LIN {X 0,Y 227.878,Z 329.572,A -85,B 0,C 180,E1 -19946.376,E2 -19946.376} C_VEL
LIN {X 0,Y 227.902,Z 329.591,A -85,B 0,C 180,E1 -19950.434,E2 -19950.434} C_VEL
LIN {X 0,Y 227.922,Z 329.564,A -85,B 0,C 180,E1 -19954.424,E2 -19954.424} C_VEL
LIN {X 0,Y 227.944,Z 329.583,A -85,B 0,C 180,E1 -19958.284,E2 -19958.284} C_VEL
LIN {X 0,Y 228.03,Z 329.545,A -85,B 0,C 180,E1 -19962.826,E2 -19962.826} C_VEL
LIN {X 0,Y 228.067,Z 329.562,A -85,B 0,C 180,E1 -19967.542,E2 -19967.542} C_VEL
LIN {X 0,Y 228.263,Z 329.504,A -85,B 0,C 180,E1 -19971.143,E2 -19971.143} C_VEL
LIN {X 0,Y 228.319,Z 329.521,A -85,B 0,C 180,E1 -19972.926,E2 -19972.926} C_VEL
LIN {X 0,Y 228.549,Z 329.485,A -85,B 0,C 180,E1 -19978.237,E2 -19978.237} C_VEL
LIN {X 0,Y 228.548,Z 329.475,A -85,B 0,C 180,E1 -19981.761,E2 -19981.761} C_VEL
LIN {X 0,Y 228.318,Z 329.531,A -85,B 0,C 180,E1 -19987.072,E2 -19987.072} C_VEL
LIN {X 0,Y 228.14,Z 329.521,A -85,B 0,C 180,E1 -19990.65,E2 -19990.65} C_VEL
LIN {X 0,Y 228.057,Z 329.576,A -85,B 0,C 180,E1 -19994.272,E2 -19994.272} C_VEL
LIN {X 0,Y 227.997,Z 329.55,A -85,B 0,C 180,E1 -19997.953,E2 -19997.953} C_VEL
LIN {X 0,Y 227.924,Z 329.589,A -85,B 0,C 180,E1 -20002.329,E2 -20002.329} C_VEL
LIN {X 0,Y 227.936,Z 329.561,A -85,B 0,C 180,E1 -20006.602,E2 -20006.602} C_VEL
LIN {X 0,Y 227.891,Z 329.596,A -85,B 0,C 180,E1 -20010.291,E2 -20010.291} C_VEL
LIN {X 0,Y 227.884,Z 329.576,A -85,B 0,C 180,E1 -20013.718,E2 -20013.718} C_VEL
LIN {X 0,Y 227.866,Z 329.604,A -85,B 0,C 180,E1 -20018.085,E2 -20018.085} C_VEL
LIN {X 0,Y 227.904,Z 329.593,A -85,B 0,C 180,E1 -20022.719,E2 -20022.719} C_VEL
LIN {X 0,Y 227.815,Z 329.543,A -85,B 0,C 180,E1 -20027.26,E2 -20027.26} C_VEL
LIN {X 0,Y 227.865,Z 329.603,A -85,B 0,C 180,E1 -20031.914,E2 -20031.914} C_VEL
LIN {X 0,Y 227.948,Z 329.901,A -85,B 0,C 180,E1 -20032.928,E2 -20032.928} C_VEL
LIN {X 0,Y 228.323,Z 331.21,A -85,B 0,C 180,E1 -20033.243,E2 -20033.243} C_VEL
LIN {X 0,Y 229.942,Z 333.723,A -85,B 0,C 180,E1 -20033.654,E2 -20033.654} C_VEL
LIN {X 0,Y 238.78,Z 348.968,A -85,B 0,C 180,E1 -20035.756,E2 -20035.756} C_VEL
LIN {X 0,Y 244.929,Z 360.706,A -85,B 0,C 180,E1 -20037.14,E2 -20037.14} C_VEL
LIN {X 0,Y 252.144,Z 374.306,A -85,B 0,C 180,E1 -20038.647,E2 -20038.647} C_VEL
LIN {X 0,Y 260.818,Z 387.178,A -85,B 0,C 180,E1 -20040.211,E2 -20040.211} C_VEL
LIN {X 0,Y 271.78,Z 400.26,A -85,B 0,C 180,E1 -20041.921,E2 -20041.921} C_VEL
LIN {X 0,Y 286.362,Z 414.958,A -85,B 0,C 180,E1 -20043.882,E2 -20043.882} C_VEL
LIN {X 0,Y 299.444,Z 426.122,A -85,B 0,C 180,E1 -20045.43,E2 -20045.43} C_VEL
LIN {X 0,Y 307.549,Z 432.734,A -85,B 0,C 180,E1 -20046.478,E2 -20046.478} C_VEL
LIN {X 0,Y 315.593,Z 438.951,A -85,B 0,C 180,E1 -20047.734,E2 -20047.734} C_VEL
LIN {X 0,Y 323.402,Z 444.777,A -85,B 0,C 180,E1 -20049.138,E2 -20049.138} C_VEL
LIN {X 0,Y 331.993,Z 451.224,A -85,B 0,C 180,E1 -20050.908,E2 -20050.908} C_VEL
LIN {X 0,Y 339.546,Z 456.264,A -85,B 0,C 180,E1 -20052.64,E2 -20052.64} C_VEL
LIN {X 0,Y 346.066,Z 461.128,A -85,B 0,C 180,E1 -20054.389,E2 -20054.389} C_VEL
LIN {X 0,Y 351.939,Z 464.834,A -85,B 0,C 180,E1 -20056.135,E2 -20056.135} C_VEL
LIN {X 0,Y 355.953,Z 467.098,A -85,B 0,C 180,E1 -20057.457,E2 -20057.457} C_VEL
LIN {X 0,Y 359.121,Z 469.614,A -85,B 0,C 180,E1 -20058.715,E2 -20058.715} C_VEL
LIN {X 0,Y 363.316,Z 472.458,A -85,B 0,C 180,E1 -20060.586,E2 -20060.586} C_VEL
LIN {X 0,Y 366.572,Z 474.299,A -85,B 0,C 180,E1 -20062.288,E2 -20062.288} C_VEL
LIN {X 0,Y 368.408,Z 475.23,A -85,B 0,C 180,E1 -20063.428,E2 -20063.428} C_VEL
LIN {X 0,Y 369.974,Z 475.879,A -85,B 0,C 180,E1 -20064.55,E2 -20064.55} C_VEL
LIN {X 0,Y 371.244,Z 476.349,A -85,B 0,C 180,E1 -20065.657,E2 -20065.657} C_VEL
LIN {X 0,Y 372.236,Z 476.635,A -85,B 0,C 180,E1 -20066.753,E2 -20066.753} C_VEL
LIN {X 0,Y 372.866,Z 477.016,A -85,B 0,C 180,E1 -20067.84,E2 -20067.84} C_VEL
LIN {X 0,Y 373.24,Z 477.247,A -85,B 0,C 180,E1 -20068.921,E2 -20068.921} C_VEL
LIN {X 0,Y 373.406,Z 477.203,A -85,B 0,C 180,E1 -20070,E2 -20070} C_VEL
LIN {X 0,Y 373.262,Z 477.182,A -85,B 0,C 180,E1 -20071.079,E2 -20071.079} C_VEL
LIN {X 0,Y 372.799,Z 476.9,A -85,B 0,C 180,E1 -20072.374,E2 -20072.374} C_VEL
LIN {X 0,Y 371.247,Z 476.345,A -85,B 0,C 180,E1 -20074.343,E2 -20074.343} C_VEL
LIN {X 0,Y 369.982,Z 475.883,A -85,B 0,C 180,E1 -20075.45,E2 -20075.45} C_VEL
LIN {X 0,Y 368.059,Z 475.041,A -85,B 0,C 180,E1 -20076.825,E2 -20076.825} C_VEL
LIN {X 0,Y 366.576,Z 474.352,A -85,B 0,C 180,E1 -20077.712,E2 -20077.712} C_VEL
LIN {X 0,Y 363.307,Z 472.462,A -85,B 0,C 180,E1 -20079.406,E2 -20079.406} C_VEL
LIN {X 0,Y 359.105,Z 469.613,A -85,B 0,C 180,E1 -20081.286,E2 -20081.286} C_VEL
LIN {X 0,Y 355.912,Z 467.07,A -85,B 0,C 180,E1 -20082.545,E2 -20082.545} C_VEL
LIN {X 0,Y 351.918,Z 464.861,A -85,B 0,C 180,E1 -20083.865,E2 -20083.865} C_VEL
LIN {X 0,Y 345.56,Z 460.756,A -85,B 0,C 180,E1 -20085.755,E2 -20085.755} C_VEL
LIN {X 0,Y 338.472,Z 455.62,A -85,B 0,C 180,E1 -20087.612,E2 -20087.612} C_VEL
LIN {X 0,Y 330.629,Z 450.246,A -85,B 0,C 180,E1 -20089.388,E2 -20089.388} C_VEL
LIN {X 0,Y 323.191,Z 444.661,A -85,B 0,C 180,E1 -20090.898,E2 -20090.898} C_VEL
LIN {X 0,Y 315.18,Z 438.628,A -85,B 0,C 180,E1 -20092.332,E2 -20092.332} C_VEL
LIN {X 0,Y 306.65,Z 432.052,A -85,B 0,C 180,E1 -20093.65,E2 -20093.65} C_VEL
LIN {X 0,Y 297.197,Z 424.33,A -85,B 0,C 180,E1 -20094.843,E2 -20094.843} C_VEL
LIN {X 0,Y 282.743,Z 411.497,A -85,B 0,C 180,E1 -20096.577,E2 -20096.577} C_VEL
LIN {X 0,Y 269.021,Z 397.22,A -85,B 0,C 180,E1 -20098.486,E2 -20098.486} C_VEL
LIN {X 0,Y 260.299,Z 386.445,A -85,B 0,C 180,E1 -20099.878,E2 -20099.878} C_VEL
LIN {X 0,Y 252.01,Z 374.071,A -85,B 0,C 180,E1 -20101.38,E2 -20101.38} C_VEL
LIN {X 0,Y 245.107,Z 361.073,A -85,B 0,C 180,E1 -20102.82,E2 -20102.82} C_VEL
LIN {X 0,Y 239.021,Z 349.422,A -85,B 0,C 180,E1 -20104.188,E2 -20104.188} C_VEL
LIN {X 0,Y 231.592,Z 336.596,A -85,B 0,C 180,E1 -20105.936,E2 -20105.936} C_VEL
LIN {X 0,Y 229.583,Z 333.337,A -85,B 0,C 180,E1 -20106.427,E2 -20106.427} C_VEL
LIN {X 0,Y 228.039,Z 330.419,A -85,B 0,C 180,E1 -20106.894,E2 -20106.894} C_VEL
LIN {X 0,Y 227.9,Z 329.657,A -85,B 0,C 180,E1 -20107.311,E2 -20107.311} C_VEL
LIN {X 0,Y 227.83,Z 329.551,A -85,B 0,C 180,E1 -20110.375,E2 -20110.375} C_VEL
LIN {X 0,Y 227.852,Z 329.579,A -85,B 0,C 180,E1 -20115.187,E2 -20115.187} C_VEL
LIN {X 0,Y 227.904,Z 329.586,A -85,B 0,C 180,E1 -20117.739,E2 -20117.739} C_VEL
LIN {X 0,Y 227.866,Z 329.604,A -85,B 0,C 180,E1 -20121.915,E2 -20121.915} C_VEL
LIN {X 0,Y 227.884,Z 329.576,A -85,B 0,C 180,E1 -20126.374,E2 -20126.374} C_VEL
LIN {X 0,Y 227.898,Z 329.583,A -85,B 0,C 180,E1 -20130.436,E2 -20130.436} C_VEL
LIN {X 0,Y 227.923,Z 329.574,A -85,B 0,C 180,E1 -20134.426,E2 -20134.426} C_VEL
LIN {X 0,Y 227.956,Z 329.575,A -85,B 0,C 180,E1 -20138.288,E2 -20138.288} C_VEL
LIN {X 0,Y 228.029,Z 329.557,A -85,B 0,C 180,E1 -20142.827,E2 -20142.827} C_VEL
LIN {X 0,Y 228.066,Z 329.554,A -85,B 0,C 180,E1 -20147.544,E2 -20147.544} C_VEL
LIN {X 0,Y 228.261,Z 329.51,A -85,B 0,C 180,E1 -20151.145,E2 -20151.145} C_VEL
LIN {X 0,Y 228.318,Z 329.531,A -85,B 0,C 180,E1 -20152.928,E2 -20152.928} C_VEL
LIN {X 0,Y 228.548,Z 329.475,A -85,B 0,C 180,E1 -20158.239,E2 -20158.239} C_VEL
LIN {X 0,Y 228.549,Z 329.485,A -85,B 0,C 180,E1 -20161.763,E2 -20161.763} C_VEL
LIN {X 0,Y 228.319,Z 329.521,A -85,B 0,C 180,E1 -20167.074,E2 -20167.074} C_VEL
LIN {X 0,Y 228.141,Z 329.523,A -85,B 0,C 180,E1 -20170.652,E2 -20170.652} C_VEL
LIN {X 0,Y 228.056,Z 329.575,A -85,B 0,C 180,E1 -20174.274,E2 -20174.274} C_VEL
LIN {X 0,Y 227.998,Z 329.542,A -85,B 0,C 180,E1 -20177.955,E2 -20177.955} C_VEL
LIN {X 0,Y 227.914,Z 329.591,A -85,B 0,C 180,E1 -20182.322,E2 -20182.322} C_VEL
LIN {X 0,Y 227.939,Z 329.556,A -85,B 0,C 180,E1 -20186.603,E2 -20186.603} C_VEL
LIN {X 0,Y 227.895,Z 329.597,A -85,B 0,C 180,E1 -20190.292,E2 -20190.292} C_VEL
LIN {X 0,Y 227.876,Z 329.572,A -85,B 0,C 180,E1 -20193.722,E2 -20193.722} C_VEL
LIN {X 0,Y 227.842,Z 329.599,A -85,B 0,C 180,E1 -20198.093,E2 -20198.093} C_VEL
LIN {X 0,Y 227.803,Z 329.608,A -85,B 0,C 180,E1 -20202.746,E2 -20202.746} C_VEL
LIN {X 0,Y 227.825,Z 329.62,A -85,B 0,C 180,E1 -20207.425,E2 -20207.425} C_VEL
LIN {X 0,Y 229.604,Z 337.052,A -85,B 0,C 180,E1 -20212.253,E2 -20212.253} C_VEL
LIN {X 0,Y 230.128,Z 339.355,A -85,B 0,C 180,E1 -20213.453,E2 -20213.453} C_VEL
LIN {X 0,Y 232.001,Z 343.344,A -85,B 0,C 180,E1 -20214.006,E2 -20214.006} C_VEL
LIN {X 0,Y 238.477,Z 356.937,A -85,B 0,C 180,E1 -20215.607,E2 -20215.607} C_VEL
LIN {X 0,Y 243.683,Z 369.149,A -85,B 0,C 180,E1 -20216.856,E2 -20216.856} C_VEL
LIN {X 0,Y 247.391,Z 390.036,A -85,B 0,C 180,E1 -20218.112,E2 -20218.112} C_VEL
LIN {X 0,Y 248.128,Z 394.813,A -85,B 0,C 180,E1 -20218.376,E2 -20218.376} C_VEL
LIN {X 0,Y 248.036,Z 398.357,A -85,B 0,C 180,E1 -20218.48,E2 -20218.48} C_VEL
LIN {X 0,Y 247.212,Z 404.208,A -85,B 0,C 180,E1 -20218.559,E2 -20218.559} C_VEL
LIN {X 0,Y 241.542,Z 423.223,A -85,B 0,C 180,E1 -20218.39,E2 -20218.39} C_VEL
LIN {X 0,Y 240.791,Z 429.07,A -85,B 0,C 180,E1 -20218.481,E2 -20218.481} C_VEL
LIN {X 0,Y 239.894,Z 448.706,A -85,B 0,C 180,E1 -20219.122,E2 -20219.122} C_VEL
LIN {X 0,Y 238.364,Z 462.733,A -85,B 0,C 180,E1 -20219.919,E2 -20219.919} C_VEL
LIN {X 0,Y 236.772,Z 473.371,A -85,B 0,C 180,E1 -20220.798,E2 -20220.798} C_VEL
LIN {X 0,Y 234.904,Z 483.507,A -85,B 0,C 180,E1 -20221.887,E2 -20221.887} C_VEL
LIN {X 0,Y 232.976,Z 492.498,A -85,B 0,C 180,E1 -20223.097,E2 -20223.097} C_VEL
LIN {X 0,Y 230.911,Z 501.222,A -85,B 0,C 180,E1 -20224.539,E2 -20224.539} C_VEL
LIN {X 0,Y 228.989,Z 508.613,A -85,B 0,C 180,E1 -20226.005,E2 -20226.005} C_VEL
LIN {X 0,Y 227.036,Z 515.83,A -85,B 0,C 180,E1 -20227.716,E2 -20227.716} C_VEL
LIN {X 0,Y 225.39,Z 522.16,A -85,B 0,C 180,E1 -20229.508,E2 -20229.508} C_VEL
LIN {X 0,Y 223.506,Z 528.569,A -85,B 0,C 180,E1 -20231.673,E2 -20231.673} C_VEL
LIN {X 0,Y 222.258,Z 533.072,A -85,B 0,C 180,E1 -20233.466,E2 -20233.466} C_VEL
LIN {X 0,Y 220.614,Z 538.563,A -85,B 0,C 180,E1 -20236.177,E2 -20236.177} C_VEL
LIN {X 0,Y 219.59,Z 542.893,A -85,B 0,C 180,E1 -20238.929,E2 -20238.929} C_VEL
LIN {X 0,Y 219.09,Z 545.263,A -85,B 0,C 180,E1 -20240.771,E2 -20240.771} C_VEL
LIN {X 0,Y 218.738,Z 547.065,A -85,B 0,C 180,E1 -20242.616,E2 -20242.616} C_VEL
LIN {X 0,Y 218.501,Z 549.519,A -85,B 0,C 180,E1 -20246.312,E2 -20246.312} C_VEL
LIN {X 0,Y 218.525,Z 550.112,A -85,B 0,C 180,E1 -20248.157,E2 -20248.157} C_VEL
LIN {X 0,Y 218.623,Z 550.27,A -85,B 0,C 180,E1 -20250,E2 -20250} C_VEL
LIN {X 0,Y 218.524,Z 550.112,A -85,B 0,C 180,E1 -20251.843,E2 -20251.843} C_VEL
LIN {X 0,Y 218.484,Z 549.256,A -85,B 0,C 180,E1 -20254.292,E2 -20254.292} C_VEL
LIN {X 0,Y 218.711,Z 547.064,A -85,B 0,C 180,E1 -20257.385,E2 -20257.385} C_VEL
LIN {X 0,Y 219.319,Z 544.111,A -85,B 0,C 180,E1 -20260.151,E2 -20260.151} C_VEL
LIN {X 0,Y 220.226,Z 540.118,A -85,B 0,C 180,E1 -20262.908,E2 -20262.908} C_VEL
LIN {X 0,Y 221.657,Z 534.987,A -85,B 0,C 180,E1 -20265.635,E2 -20265.635} C_VEL
LIN {X 0,Y 223.184,Z 529.726,A -85,B 0,C 180,E1 -20267.88,E2 -20267.88} C_VEL
LIN {X 0,Y 225.063,Z 523.411,A -85,B 0,C 180,E1 -20270.089,E2 -20270.089} C_VEL
LIN {X 0,Y 226.621,Z 517.457,A -85,B 0,C 180,E1 -20271.847,E2 -20271.847} C_VEL
LIN {X 0,Y 228.474,Z 510.531,A -85,B 0,C 180,E1 -20273.571,E2 -20273.571} C_VEL
LIN {X 0,Y 230.658,Z 502.357,A -85,B 0,C 180,E1 -20275.249,E2 -20275.249} C_VEL
LIN {X 0,Y 232.662,Z 493.849,A -85,B 0,C 180,E1 -20276.7,E2 -20276.7} C_VEL
LIN {X 0,Y 234.592,Z 485.139,A -85,B 0,C 180,E1 -20277.91,E2 -20277.91} C_VEL
LIN {X 0,Y 236.374,Z 475.383,A -85,B 0,C 180,E1 -20279.012,E2 -20279.012} C_VEL
LIN {X 0,Y 237.76,Z 466.593,A -85,B 0,C 180,E1 -20279.799,E2 -20279.799} C_VEL
LIN {X 0,Y 239.164,Z 456.049,A -85,B 0,C 180,E1 -20280.5,E2 -20280.5} C_VEL
LIN {X 0,Y 240.048,Z 446.427,A -85,B 0,C 180,E1 -20280.96,E2 -20280.96} C_VEL
LIN {X 0,Y 241.421,Z 414.37,A -85,B 0,C 180,E1 -20281.93,E2 -20281.93} C_VEL
LIN {X 0,Y 242.009,Z 395.189,A -85,B 0,C 180,E1 -20282.501,E2 -20282.501} C_VEL
LIN {X 0,Y 238.137,Z 372.45,A -85,B 0,C 180,E1 -20283.896,E2 -20283.896} C_VEL
LIN {X 0,Y 232.185,Z 358.251,A -85,B 0,C 180,E1 -20285.406,E2 -20285.406} C_VEL
LIN {X 0,Y 224.648,Z 342.853,A -85,B 0,C 180,E1 -20287.378,E2 -20287.378} C_VEL
LIN {X 0,Y 222.799,Z 338.923,A -85,B 0,C 180,E1 -20288.001,E2 -20288.001} C_VEL
LIN {X 0,Y 221.282,Z 332.871,A -85,B 0,C 180,E1 -20291.832,E2 -20291.832} C_VEL
LIN {X 0,Y 220.752,Z 330.49,A -85,B 0,C 180,E1 -20293.611,E2 -20293.611} C_VEL
LIN {X 0,Y 220.762,Z 330.485,A -85,B 0,C 180,E1 -20298.044,E2 -20298.044} C_VEL
LIN {X 0,Y 220.824,Z 330.479,A -85,B 0,C 180,E1 -20302.792,E2 -20302.792} C_VEL
LIN {X 0,Y 220.815,Z 330.458,A -85,B 0,C 180,E1 -20307.242,E2 -20307.242} C_VEL
LIN {X 0,Y 220.824,Z 330.454,A -85,B 0,C 180,E1 -20311.484,E2 -20311.484} C_VEL
LIN {X 0,Y 220.859,Z 330.46,A -85,B 0,C 180,E1 -20315.563,E2 -20315.563} C_VEL
LIN {X 0,Y 220.88,Z 330.442,A -85,B 0,C 180,E1 -20319.512,E2 -20319.512} C_VEL
LIN {X 0,Y 221.011,Z 330.426,A -85,B 0,C 180,E1 -20323.369,E2 -20323.369} C_VEL
LIN {X 0,Y 221.006,Z 330.445,A -85,B 0,C 180,E1 -20327.137,E2 -20327.137} C_VEL
LIN {X 0,Y 221.2,Z 330.382,A -85,B 0,C 180,E1 -20330.858,E2 -20330.858} C_VEL
LIN {X 0,Y 221.254,Z 330.395,A -85,B 0,C 180,E1 -20332.699,E2 -20332.699} C_VEL
LIN {X 0,Y 221.507,Z 330.361,A -85,B 0,C 180,E1 -20338.181,E2 -20338.181} C_VEL
LIN {X 0,Y 221.506,Z 330.352,A -85,B 0,C 180,E1 -20341.817,E2 -20341.817} C_VEL
LIN {X 0,Y 221.253,Z 330.407,A -85,B 0,C 180,E1 -20347.299,E2 -20347.299} C_VEL
LIN {X 0,Y 221.062,Z 330.404,A -85,B 0,C 180,E1 -20350.996,E2 -20350.996} C_VEL
LIN {X 0,Y 220.989,Z 330.459,A -85,B 0,C 180,E1 -20354.738,E2 -20354.738} C_VEL
LIN {X 0,Y 220.916,Z 330.427,A -85,B 0,C 180,E1 -20358.549,E2 -20358.549} C_VEL
LIN {X 0,Y 220.891,Z 330.467,A -85,B 0,C 180,E1 -20362.682,E2 -20362.682} C_VEL
LIN {X 0,Y 220.878,Z 330.437,A -85,B 0,C 180,E1 -20367.014,E2 -20367.014} C_VEL
LIN {X 0,Y 220.833,Z 330.478,A -85,B 0,C 180,E1 -20370.767,E2 -20370.767} C_VEL
LIN {X 0,Y 220.81,Z 330.454,A -85,B 0,C 180,E1 -20374.952,E2 -20374.952} C_VEL
LIN {X 0,Y 220.851,Z 330.459,A -85,B 0,C 180,E1 -20379.526,E2 -20379.526} C_VEL
LIN {X 0,Y 220.861,Z 330.472,A -85,B 0,C 180,E1 -20382.957,E2 -20382.957} C_VEL
LIN {X 0,Y 220.774,Z 330.417,A -85,B 0,C 180,E1 -20388.05,E2 -20388.05} C_VEL
LIN {X 0,Y 220.834,Z 330.704,A -85,B 0,C 180,E1 -20391.492,E2 -20391.492} C_VEL
LIN {X 0,Y 221.134,Z 331.799,A -85,B 0,C 180,E1 -20391.846,E2 -20391.846} C_VEL
LIN {X 0,Y 222.663,Z 334.447,A -85,B 0,C 180,E1 -20392.282,E2 -20392.282} C_VEL
LIN {X 0,Y 223.911,Z 336.348,A -85,B 0,C 180,E1 -20392.606,E2 -20392.606} C_VEL
LIN {X 0,Y 230.101,Z 346.534,A -85,B 0,C 180,E1 -20394.169,E2 -20394.169} C_VEL
LIN {X 0,Y 237.952,Z 360.997,A -85,B 0,C 180,E1 -20396.05,E2 -20396.05} C_VEL
LIN {X 0,Y 246.369,Z 377.37,A -85,B 0,C 180,E1 -20397.922,E2 -20397.922} C_VEL
LIN {X 0,Y 254.153,Z 389.318,A -85,B 0,C 180,E1 -20399.409,E2 -20399.409} C_VEL
LIN {X 0,Y 261.639,Z 398.978,A -85,B 0,C 180,E1 -20400.68,E2 -20400.68} C_VEL
LIN {X 0,Y 273.729,Z 412.316,A -85,B 0,C 180,E1 -20402.491,E2 -20402.491} C_VEL
LIN {X 0,Y 285.746,Z 423.639,A -85,B 0,C 180,E1 -20404.059,E2 -20404.059} C_VEL
LIN {X 0,Y 296.322,Z 432.546,A -85,B 0,C 180,E1 -20405.321,E2 -20405.321} C_VEL
LIN {X 0,Y 304.747,Z 439.439,A -85,B 0,C 180,E1 -20406.447,E2 -20406.447} C_VEL
LIN {X 0,Y 312.979,Z 445.791,A -85,B 0,C 180,E1 -20407.749,E2 -20407.749} C_VEL
LIN {X 0,Y 321.068,Z 451.705,A -85,B 0,C 180,E1 -20409.206,E2 -20409.206} C_VEL
LIN {X 0,Y 329.282,Z 457.928,A -85,B 0,C 180,E1 -20410.918,E2 -20410.918} C_VEL
LIN {X 0,Y 335.929,Z 462.269,A -85,B 0,C 180,E1 -20412.432,E2 -20412.432} C_VEL
LIN {X 0,Y 343.054,Z 467.541,A -85,B 0,C 180,E1 -20414.335,E2 -20414.335} C_VEL
LIN {X 0,Y 348.712,Z 471.122,A -85,B 0,C 180,E1 -20416.005,E2 -20416.005} C_VEL
LIN {X 0,Y 352.903,Z 473.494,A -85,B 0,C 180,E1 -20417.372,E2 -20417.372} C_VEL
LIN {X 0,Y 357.621,Z 477.083,A -85,B 0,C 180,E1 -20419.293,E2 -20419.293} C_VEL
LIN {X 0,Y 361.361,Z 479.527,A -85,B 0,C 180,E1 -20421.049,E2 -20421.049} C_VEL
LIN {X 0,Y 363.554,Z 480.72,A -85,B 0,C 180,E1 -20422.223,E2 -20422.223} C_VEL
LIN {X 0,Y 365.437,Z 481.66,A -85,B 0,C 180,E1 -20423.374,E2 -20423.374} C_VEL
LIN {X 0,Y 367.106,Z 482.343,A -85,B 0,C 180,E1 -20424.558,E2 -20424.558} C_VEL
LIN {X 0,Y 368.313,Z 482.82,A -85,B 0,C 180,E1 -20425.623,E2 -20425.623} C_VEL
LIN {X 0,Y 369.336,Z 483.098,A -85,B 0,C 180,E1 -20426.728,E2 -20426.728} C_VEL
LIN {X 0,Y 369.975,Z 483.474,A -85,B 0,C 180,E1 -20427.823,E2 -20427.823} C_VEL
LIN {X 0,Y 370.339,Z 483.726,A -85,B 0,C 180,E1 -20428.913,E2 -20428.913} C_VEL
LIN {X 0,Y 370.525,Z 483.663,A -85,B 0,C 180,E1 -20430,E2 -20430} C_VEL
LIN {X 0,Y 370.371,Z 483.642,A -85,B 0,C 180,E1 -20431.087,E2 -20431.087} C_VEL
LIN {X 0,Y 369.987,Z 483.423,A -85,B 0,C 180,E1 -20432.177,E2 -20432.177} C_VEL
LIN {X 0,Y 369.321,Z 483.102,A -85,B 0,C 180,E1 -20433.273,E2 -20433.273} C_VEL
LIN {X 0,Y 368.31,Z 482.8,A -85,B 0,C 180,E1 -20434.377,E2 -20434.377} C_VEL
LIN {X 0,Y 367.031,Z 482.313,A -85,B 0,C 180,E1 -20435.494,E2 -20435.494} C_VEL
LIN {X 0,Y 365.444,Z 481.652,A -85,B 0,C 180,E1 -20436.626,E2 -20436.626} C_VEL
LIN {X 0,Y 362.343,Z 480.064,A -85,B 0,C 180,E1 -20438.435,E2 -20438.435} C_VEL
LIN {X 0,Y 358.865,Z 477.939,A -85,B 0,C 180,E1 -20440.151,E2 -20440.151} C_VEL
LIN {X 0,Y 354.945,Z 475.149,A -85,B 0,C 180,E1 -20441.816,E2 -20441.816} C_VEL
LIN {X 0,Y 352.819,Z 473.432,A -85,B 0,C 180,E1 -20442.657,E2 -20442.657} C_VEL
LIN {X 0,Y 347.994,Z 470.716,A -85,B 0,C 180,E1 -20444.215,E2 -20444.215} C_VEL
LIN {X 0,Y 343.051,Z 467.515,A -85,B 0,C 180,E1 -20445.664,E2 -20445.664} C_VEL
LIN {X 0,Y 338.092,Z 463.919,A -85,B 0,C 180,E1 -20447.021,E2 -20447.021} C_VEL
LIN {X 0,Y 330.724,Z 458.91,A -85,B 0,C 180,E1 -20448.764,E2 -20448.764} C_VEL
LIN {X 0,Y 323.285,Z 453.33,A -85,B 0,C 180,E1 -20450.354,E2 -20450.354} C_VEL
LIN {X 0,Y 314.631,Z 447.083,A -85,B 0,C 180,E1 -20451.967,E2 -20451.967} C_VEL
LIN {X 0,Y 306.173,Z 440.522,A -85,B 0,C 180,E1 -20453.342,E2 -20453.342} C_VEL
LIN {X 0,Y 298.373,Z 434.289,A -85,B 0,C 180,E1 -20454.424,E2 -20454.424} C_VEL
LIN {X 0,Y 286.312,Z 424.127,A -85,B 0,C 180,E1 -20455.872,E2 -20455.872} C_VEL
LIN {X 0,Y 276.694,Z 415.179,A -85,B 0,C 180,E1 -20457.106,E2 -20457.106} C_VEL
LIN {X 0,Y 264.358,Z 402.242,A -85,B 0,C 180,E1 -20458.887,E2 -20458.887} C_VEL
LIN {X 0,Y 255.511,Z 391.242,A -85,B 0,C 180,E1 -20460.348,E2 -20460.348} C_VEL
LIN {X 0,Y 247.05,Z 378.539,A -85,B 0,C 180,E1 -20461.939,E2 -20461.939} C_VEL
LIN {X 0,Y 240.025,Z 365.188,A -85,B 0,C 180,E1 -20463.467,E2 -20463.467} C_VEL
LIN {X 0,Y 232.852,Z 351.396,A -85,B 0,C 180,E1 -20465.16,E2 -20465.16} C_VEL
LIN {X 0,Y 225.32,Z 338.515,A -85,B 0,C 180,E1 -20467.034,E2 -20467.034} C_VEL
LIN {X 0,Y 222.666,Z 334.413,A -85,B 0,C 180,E1 -20467.718,E2 -20467.718} C_VEL
LIN {X 0,Y 221.134,Z 331.801,A -85,B 0,C 180,E1 -20468.154,E2 -20468.154} C_VEL
LIN {X 0,Y 220.855,Z 330.69,A -85,B 0,C 180,E1 -20468.515,E2 -20468.515} C_VEL
LIN {X 0,Y 220.774,Z 330.417,A -85,B 0,C 180,E1 -20471.95,E2 -20471.95} C_VEL
LIN {X 0,Y 220.861,Z 330.472,A -85,B 0,C 180,E1 -20477.043,E2 -20477.043} C_VEL
LIN {X 0,Y 220.851,Z 330.459,A -85,B 0,C 180,E1 -20480.474,E2 -20480.474} C_VEL
LIN {X 0,Y 220.81,Z 330.454,A -85,B 0,C 180,E1 -20485.048,E2 -20485.048} C_VEL
LIN {X 0,Y 220.828,Z 330.477,A -85,B 0,C 180,E1 -20489.39,E2 -20489.39} C_VEL
LIN {X 0,Y 220.889,Z 330.439,A -85,B 0,C 180,E1 -20493.55,E2 -20493.55} C_VEL
LIN {X 0,Y 220.872,Z 330.468,A -85,B 0,C 180,E1 -20497.554,E2 -20497.554} C_VEL
LIN {X 0,Y 220.979,Z 330.43,A -85,B 0,C 180,E1 -20502.572,E2 -20502.572} C_VEL
LIN {X 0,Y 221.005,Z 330.441,A -85,B 0,C 180,E1 -20507.139,E2 -20507.139} C_VEL
LIN {X 0,Y 221.199,Z 330.386,A -85,B 0,C 180,E1 -20510.86,E2 -20510.86} C_VEL
LIN {X 0,Y 221.253,Z 330.407,A -85,B 0,C 180,E1 -20512.701,E2 -20512.701} C_VEL
LIN {X 0,Y 221.506,Z 330.352,A -85,B 0,C 180,E1 -20518.183,E2 -20518.183} C_VEL
LIN {X 0,Y 221.507,Z 330.361,A -85,B 0,C 180,E1 -20521.819,E2 -20521.819} C_VEL
LIN {X 0,Y 221.254,Z 330.395,A -85,B 0,C 180,E1 -20527.301,E2 -20527.301} C_VEL
LIN {X 0,Y 221.063,Z 330.408,A -85,B 0,C 180,E1 -20530.998,E2 -20530.998} C_VEL
LIN {X 0,Y 220.988,Z 330.453,A -85,B 0,C 180,E1 -20534.74,E2 -20534.74} C_VEL
LIN {X 0,Y 220.916,Z 330.422,A -85,B 0,C 180,E1 -20538.551,E2 -20538.551} C_VEL
LIN {X 0,Y 220.882,Z 330.47,A -85,B 0,C 180,E1 -20542.676,E2 -20542.676} C_VEL
LIN {X 0,Y 220.88,Z 330.435,A -85,B 0,C 180,E1 -20547.015,E2 -20547.015} C_VEL
LIN {X 0,Y 220.837,Z 330.477,A -85,B 0,C 180,E1 -20550.769,E2 -20550.769} C_VEL
LIN {X 0,Y 220.8,Z 330.457,A -85,B 0,C 180,E1 -20554.956,E2 -20554.956} C_VEL
LIN {X 0,Y 220.809,Z 330.481,A -85,B 0,C 180,E1 -20557.28,E2 -20557.28} C_VEL
LIN {X 0,Y 220.762,Z 330.485,A -85,B 0,C 180,E1 -20561.956,E2 -20561.956} C_VEL
LIN {X 0,Y 220.752,Z 330.521,A -85,B 0,C 180,E1 -20566.494,E2 -20566.494} C_VEL
LIN {X 0,Y 222.588,Z 338.246,A -85,B 0,C 180,E1 -20571.665,E2 -20571.665} C_VEL
LIN {X 0,Y 222.964,Z 339.52,A -85,B 0,C 180,E1 -20572.125,E2 -20572.125} C_VEL
LIN {X 0,Y 229.857,Z 353.313,A -85,B 0,C 180,E1 -20573.997,E2 -20573.997} C_VEL
LIN {X 0,Y 236.283,Z 367.626,A -85,B 0,C 180,E1 -20575.63,E2 -20575.63} C_VEL
LIN {X 0,Y 238.272,Z 373.153,A -85,B 0,C 180,E1 -20576.151,E2 -20576.151} C_VEL
LIN {X 0,Y 241.904,Z 394.781,A -85,B 0,C 180,E1 -20577.469,E2 -20577.469} C_VEL
LIN {X 0,Y 241.924,Z 400.099,A -85,B 0,C 180,E1 -20577.655,E2 -20577.655} C_VEL
LIN {X 0,Y 240.791,Z 429.07,A -85,B 0,C 180,E1 -20578.481,E2 -20578.481} C_VEL
LIN {X 0,Y 240.025,Z 434.912,A -85,B 0,C 180,E1 -20578.568,E2 -20578.568} C_VEL
LIN {X 0,Y 237.089,Z 444.387,A -85,B 0,C 180,E1 -20578.513,E2 -20578.513} C_VEL
LIN {X 0,Y 233.878,Z 453.78,A -85,B 0,C 180,E1 -20578.573,E2 -20578.573} C_VEL
LIN {X 0,Y 232.686,Z 459.495,A -85,B 0,C 180,E1 -20578.822,E2 -20578.822} C_VEL
LIN {X 0,Y 230.782,Z 472.171,A -85,B 0,C 180,E1 -20579.837,E2 -20579.837} C_VEL
LIN {X 0,Y 228.976,Z 481.681,A -85,B 0,C 180,E1 -20580.84,E2 -20580.84} C_VEL
LIN {X 0,Y 227.007,Z 490.954,A -85,B 0,C 180,E1 -20582.079,E2 -20582.079} C_VEL
LIN {X 0,Y 224.78,Z 499.893,A -85,B 0,C 180,E1 -20583.543,E2 -20583.543} C_VEL
LIN {X 0,Y 222.497,Z 508.418,A -85,B 0,C 180,E1 -20585.259,E2 -20585.259} C_VEL
LIN {X 0,Y 220.448,Z 515.635,A -85,B 0,C 180,E1 -20587.013,E2 -20587.013} C_VEL
LIN {X 0,Y 218.785,Z 521.464,A -85,B 0,C 180,E1 -20588.682,E2 -20588.682} C_VEL
LIN {X 0,Y 216.755,Z 528.375,A -85,B 0,C 180,E1 -20591.081,E2 -20591.081} C_VEL
LIN {X 0,Y 215.451,Z 532.878,A -85,B 0,C 180,E1 -20592.928,E2 -20592.928} C_VEL
LIN {X 0,Y 213.699,Z 538.368,A -85,B 0,C 180,E1 -20595.721,E2 -20595.721} C_VEL
LIN {X 0,Y 212.579,Z 542.697,A -85,B 0,C 180,E1 -20598.559,E2 -20598.559} C_VEL
LIN {X 0,Y 212.064,Z 545.068,A -85,B 0,C 180,E1 -20600.462,E2 -20600.462} C_VEL
LIN {X 0,Y 211.493,Z 548.263,A -85,B 0,C 180,E1 -20604.279,E2 -20604.279} C_VEL
LIN {X 0,Y 211.42,Z 549.326,A -85,B 0,C 180,E1 -20606.188,E2 -20606.188} C_VEL
LIN {X 0,Y 211.427,Z 549.918,A -85,B 0,C 180,E1 -20608.095,E2 -20608.095} C_VEL
LIN {X 0,Y 211.539,Z 550.077,A -85,B 0,C 180,E1 -20610,E2 -20610} C_VEL
LIN {X 0,Y 211.426,Z 549.918,A -85,B 0,C 180,E1 -20611.905,E2 -20611.905} C_VEL
LIN {X 0,Y 211.396,Z 549.209,A -85,B 0,C 180,E1 -20614.145,E2 -20614.145} C_VEL
LIN {X 0,Y 211.652,Z 546.869,A -85,B 0,C 180,E1 -20617.632,E2 -20617.632} C_VEL
LIN {X 0,Y 212.305,Z 543.916,A -85,B 0,C 180,E1 -20620.49,E2 -20620.49} C_VEL
LIN {X 0,Y 213.261,Z 539.923,A -85,B 0,C 180,E1 -20623.337,E2 -20623.337} C_VEL
LIN {X 0,Y 214.789,Z 534.792,A -85,B 0,C 180,E1 -20626.148,E2 -20626.148} C_VEL
LIN {X 0,Y 216.389,Z 529.53,A -85,B 0,C 180,E1 -20628.461,E2 -20628.461} C_VEL
LIN {X 0,Y 218.389,Z 523.216,A -85,B 0,C 180,E1 -20630.731,E2 -20630.731} C_VEL
LIN {X 0,Y 220.011,Z 517.263,A -85,B 0,C 180,E1 -20632.539,E2 -20632.539} C_VEL
LIN {X 0,Y 221.98,Z 510.337,A -85,B 0,C 180,E1 -20634.304,E2 -20634.304} C_VEL
LIN {X 0,Y 224.239,Z 502.163,A -85,B 0,C 180,E1 -20636.025,E2 -20636.025} C_VEL
LIN {X 0,Y 226.341,Z 493.655,A -85,B 0,C 180,E1 -20637.508,E2 -20637.508} C_VEL
LIN {X 0,Y 228.319,Z 484.944,A -85,B 0,C 180,E1 -20638.747,E2 -20638.747} C_VEL
LIN {X 0,Y 230.185,Z 475.189,A -85,B 0,C 180,E1 -20639.87,E2 -20639.87} C_VEL
LIN {X 0,Y 231.629,Z 466.399,A -85,B 0,C 180,E1 -20640.671,E2 -20640.671} C_VEL
LIN {X 0,Y 233.06,Z 456.069,A -85,B 0,C 180,E1 -20641.373,E2 -20641.373} C_VEL
LIN {X 0,Y 234.021,Z 445.789,A -85,B 0,C 180,E1 -20641.871,E2 -20641.871} C_VEL
LIN {X 0,Y 235.764,Z 404.728,A -85,B 0,C 180,E1 -20643.126,E2 -20643.126} C_VEL
LIN {X 0,Y 236.002,Z 396.212,A -85,B 0,C 180,E1 -20643.392,E2 -20643.392} C_VEL
LIN {X 0,Y 232.402,Z 374.759,A -85,B 0,C 180,E1 -20644.759,E2 -20644.759} C_VEL
LIN {X 0,Y 225.766,Z 359.262,A -85,B 0,C 180,E1 -20646.525,E2 -20646.525} C_VEL
LIN {X 0,Y 219.201,Z 346.06,A -85,B 0,C 180,E1 -20648.334,E2 -20648.334} C_VEL
LIN {X 0,Y 217.067,Z 342.11,A -85,B 0,C 180,E1 -20648.942,E2 -20648.942} C_VEL
LIN {X 0,Y 215.402,Z 338.628,A -85,B 0,C 180,E1 -20649.572,E2 -20649.572} C_VEL
LIN {X 0,Y 213.758,Z 331.589,A -85,B 0,C 180,E1 -20654.347,E2 -20654.347} C_VEL
LIN {X 0,Y 213.702,Z 331.355,A -85,B 0,C 180,E1 -20656.344,E2 -20656.344} C_VEL
LIN {X 0,Y 213.708,Z 331.349,A -85,B 0,C 180,E1 -20659.144,E2 -20659.144} C_VEL
LIN {X 0,Y 213.743,Z 331.352,A -85,B 0,C 180,E1 -20663.71,E2 -20663.71} C_VEL
LIN {X 0,Y 213.766,Z 331.349,A -85,B 0,C 180,E1 -20668.261,E2 -20668.261} C_VEL
LIN {X 0,Y 213.824,Z 331.314,A -85,B 0,C 180,E1 -20672.602,E2 -20672.602} C_VEL
LIN {X 0,Y 213.817,Z 331.349,A -85,B 0,C 180,E1 -20676.973,E2 -20676.973} C_VEL
LIN {X 0,Y 213.939,Z 331.298,A -85,B 0,C 180,E1 -20682.802,E2 -20682.802} C_VEL
LIN {X 0,Y 213.947,Z 331.329,A -85,B 0,C 180,E1 -20686.705,E2 -20686.705} C_VEL
LIN {X 0,Y 214.137,Z 331.26,A -85,B 0,C 180,E1 -20690.554,E2 -20690.554} C_VEL
LIN {X 0,Y 214.096,Z 331.312,A -85,B 0,C 180,E1 -20694.347,E2 -20694.347} C_VEL
LIN {X 0,Y 214.44,Z 331.241,A -85,B 0,C 180,E1 -20698.121,E2 -20698.121} C_VEL
LIN {X 0,Y 214.541,Z 331.21,A -85,B 0,C 180,E1 -20699.999,E2 -20699.999} C_VEL
LIN {X 0,Y 214.439,Z 331.232,A -85,B 0,C 180,E1 -20701.877,E2 -20701.877} C_VEL
LIN {X 0,Y 214.193,Z 331.279,A -85,B 0,C 180,E1 -20707.541,E2 -20707.541} C_VEL
LIN {X 0,Y 213.994,Z 331.287,A -85,B 0,C 180,E1 -20711.364,E2 -20711.364} C_VEL
LIN {X 0,Y 213.927,Z 331.336,A -85,B 0,C 180,E1 -20715.236,E2 -20715.236} C_VEL
LIN {X 0,Y 213.833,Z 331.307,A -85,B 0,C 180,E1 -20719.187,E2 -20719.187} C_VEL
LIN {X 0,Y 213.842,Z 331.349,A -85,B 0,C 180,E1 -20723.226,E2 -20723.226} C_VEL
LIN {X 0,Y 213.824,Z 331.315,A -85,B 0,C 180,E1 -20727.449,E2 -20727.449} C_VEL
LIN {X 0,Y 213.764,Z 331.358,A -85,B 0,C 180,E1 -20731.737,E2 -20731.737} C_VEL
LIN {X 0,Y 213.749,Z 331.344,A -85,B 0,C 180,E1 -20736.286,E2 -20736.286} C_VEL
LIN {X 0,Y 213.789,Z 331.333,A -85,B 0,C 180,E1 -20741.106,E2 -20741.106} C_VEL
LIN {X 0,Y 213.804,Z 331.352,A -85,B 0,C 180,E1 -20743.685,E2 -20743.685} C_VEL
LIN {X 0,Y 213.714,Z 331.299,A -85,B 0,C 180,E1 -20748.876,E2 -20748.876} C_VEL
LIN {X 0,Y 213.829,Z 331.669,A -85,B 0,C 180,E1 -20750.084,E2 -20750.084} C_VEL
LIN {X 0,Y 214.157,Z 332.883,A -85,B 0,C 180,E1 -20750.406,E2 -20750.406} C_VEL
LIN {X 0,Y 215.822,Z 335.512,A -85,B 0,C 180,E1 -20750.899,E2 -20750.899} C_VEL
LIN {X 0,Y 216.935,Z 337.314,A -85,B 0,C 180,E1 -20751.214,E2 -20751.214} C_VEL
LIN {X 0,Y 223.422,Z 347.626,A -85,B 0,C 180,E1 -20752.957,E2 -20752.957} C_VEL
LIN {X 0,Y 232.271,Z 363.77,A -85,B 0,C 180,E1 -20755.197,E2 -20755.197} C_VEL
LIN {X 0,Y 241.073,Z 381.177,A -85,B 0,C 180,E1 -20757.256,E2 -20757.256} C_VEL
LIN {X 0,Y 248.857,Z 393.334,A -85,B 0,C 180,E1 -20758.813,E2 -20758.813} C_VEL
LIN {X 0,Y 256.47,Z 403.388,A -85,B 0,C 180,E1 -20760.164,E2 -20760.164} C_VEL
LIN {X 0,Y 269.631,Z 417.96,A -85,B 0,C 180,E1 -20762.199,E2 -20762.199} C_VEL
LIN {X 0,Y 281.67,Z 429.331,A -85,B 0,C 180,E1 -20763.824,E2 -20763.824} C_VEL
LIN {X 0,Y 291.894,Z 438.057,A -85,B 0,C 180,E1 -20765.148,E2 -20765.148} C_VEL
LIN {X 0,Y 301.58,Z 445.907,A -85,B 0,C 180,E1 -20766.469,E2 -20766.469} C_VEL
LIN {X 0,Y 308.411,Z 451.168,A -85,B 0,C 180,E1 -20767.538,E2 -20767.538} C_VEL
LIN {X 0,Y 316.307,Z 457,A -85,B 0,C 180,E1 -20768.936,E2 -20768.936} C_VEL
LIN {X 0,Y 323.622,Z 462.471,A -85,B 0,C 180,E1 -20770.409,E2 -20770.409} C_VEL
LIN {X 0,Y 330.8,Z 467.376,A -85,B 0,C 180,E1 -20772.007,E2 -20772.007} C_VEL
LIN {X 0,Y 337.827,Z 472.531,A -85,B 0,C 180,E1 -20773.819,E2 -20773.819} C_VEL
LIN {X 0,Y 341.974,Z 475.317,A -85,B 0,C 180,E1 -20774.994,E2 -20774.994} C_VEL
LIN {X 0,Y 346.922,Z 478.267,A -85,B 0,C 180,E1 -20776.502,E2 -20776.502} C_VEL
LIN {X 0,Y 350.596,Z 480.621,A -85,B 0,C 180,E1 -20777.782,E2 -20777.782} C_VEL
LIN {X 0,Y 355.235,Z 484.044,A -85,B 0,C 180,E1 -20779.744,E2 -20779.744} C_VEL
LIN {X 0,Y 357.774,Z 485.627,A -85,B 0,C 180,E1 -20780.959,E2 -20780.959} C_VEL
LIN {X 0,Y 361.225,Z 487.475,A -85,B 0,C 180,E1 -20782.859,E2 -20782.859} C_VEL
LIN {X 0,Y 363.585,Z 488.526,A -85,B 0,C 180,E1 -20784.454,E2 -20784.454} C_VEL
LIN {X 0,Y 364.919,Z 489.066,A -85,B 0,C 180,E1 -20785.582,E2 -20785.582} C_VEL
LIN {X 0,Y 366.043,Z 489.375,A -85,B 0,C 180,E1 -20786.741,E2 -20786.741} C_VEL
LIN {X 0,Y 366.654,Z 489.749,A -85,B 0,C 180,E1 -20787.803,E2 -20787.803} C_VEL
LIN {X 0,Y 367.034,Z 489.986,A -85,B 0,C 180,E1 -20788.903,E2 -20788.903} C_VEL
LIN {X 0,Y 367.232,Z 489.931,A -85,B 0,C 180,E1 -20790,E2 -20790} C_VEL
LIN {X 0,Y 367.068,Z 489.911,A -85,B 0,C 180,E1 -20791.097,E2 -20791.097} C_VEL
LIN {X 0,Y 366.677,Z 489.686,A -85,B 0,C 180,E1 -20792.197,E2 -20792.197} C_VEL
LIN {X 0,Y 365.979,Z 489.375,A -85,B 0,C 180,E1 -20793.303,E2 -20793.303} C_VEL
LIN {X 0,Y 364.922,Z 489.031,A -85,B 0,C 180,E1 -20794.418,E2 -20794.418} C_VEL
LIN {X 0,Y 363.566,Z 488.523,A -85,B 0,C 180,E1 -20795.546,E2 -20795.546} C_VEL
LIN {X 0,Y 361.232,Z 487.484,A -85,B 0,C 180,E1 -20797.15,E2 -20797.15} C_VEL
LIN {X 0,Y 357.794,Z 485.57,A -85,B 0,C 180,E1 -20799.041,E2 -20799.041} C_VEL
LIN {X 0,Y 353.991,Z 483.143,A -85,B 0,C 180,E1 -20800.815,E2 -20800.815} C_VEL
LIN {X 0,Y 349.072,Z 479.475,A -85,B 0,C 180,E1 -20802.795,E2 -20802.795} C_VEL
LIN {X 0,Y 344.807,Z 477.067,A -85,B 0,C 180,E1 -20804.157,E2 -20804.157} C_VEL
LIN {X 0,Y 339.967,Z 473.96,A -85,B 0,C 180,E1 -20805.589,E2 -20805.589} C_VEL
LIN {X 0,Y 334.341,Z 469.923,A -85,B 0,C 180,E1 -20807.114,E2 -20807.114} C_VEL
LIN {X 0,Y 328.781,Z 466.131,A -85,B 0,C 180,E1 -20808.449,E2 -20808.449} C_VEL
LIN {X 0,Y 321.605,Z 461.019,A -85,B 0,C 180,E1 -20810.006,E2 -20810.006} C_VEL
LIN {X 0,Y 316.304,Z 457.039,A -85,B 0,C 180,E1 -20811.063,E2 -20811.063} C_VEL
LIN {X 0,Y 308.365,Z 451.114,A -85,B 0,C 180,E1 -20812.471,E2 -20812.471} C_VEL
LIN {X 0,Y 299.592,Z 444.364,A -85,B 0,C 180,E1 -20813.813,E2 -20813.813} C_VEL
LIN {X 0,Y 286.328,Z 433.53,A -85,B 0,C 180,E1 -20815.575,E2 -20815.575} C_VEL
LIN {X 0,Y 273.074,Z 421.364,A -85,B 0,C 180,E1 -20817.319,E2 -20817.319} C_VEL
LIN {X 0,Y 259.587,Z 407.102,A -85,B 0,C 180,E1 -20819.323,E2 -20819.323} C_VEL
LIN {X 0,Y 250.585,Z 395.807,A -85,B 0,C 180,E1 -20820.865,E2 -20820.865} C_VEL
LIN {X 0,Y 242.076,Z 382.935,A -85,B 0,C 180,E1 -20822.529,E2 -20822.529} C_VEL
LIN {X 0,Y 234.986,Z 369.347,A -85,B 0,C 180,E1 -20824.138,E2 -20824.138} C_VEL
LIN {X 0,Y 228.725,Z 357.12,A -85,B 0,C 180,E1 -20825.679,E2 -20825.679} C_VEL
LIN {X 0,Y 220.913,Z 343.41,A -85,B 0,C 180,E1 -20827.709,E2 -20827.709} C_VEL
LIN {X 0,Y 216.384,Z 336.183,A -85,B 0,C 180,E1 -20828.951,E2 -20828.951} C_VEL
LIN {X 0,Y 214.254,Z 333.155,A -85,B 0,C 180,E1 -20829.554,E2 -20829.554} C_VEL
LIN {X 0,Y 213.82,Z 331.69,A -85,B 0,C 180,E1 -20829.912,E2 -20829.912} C_VEL
LIN {X 0,Y 213.718,Z 331.3,A -85,B 0,C 180,E1 -20830.859,E2 -20830.859} C_VEL
LIN {X 0,Y 213.725,Z 331.305,A -85,B 0,C 180,E1 -20833.672,E2 -20833.672} C_VEL
LIN {X 0,Y 213.807,Z 331.352,A -85,B 0,C 180,E1 -20836.349,E2 -20836.349} C_VEL
LIN {X 0,Y 213.789,Z 331.333,A -85,B 0,C 180,E1 -20839.119,E2 -20839.119} C_VEL
LIN {X 0,Y 213.749,Z 331.344,A -85,B 0,C 180,E1 -20843.714,E2 -20843.714} C_VEL
LIN {X 0,Y 213.764,Z 331.358,A -85,B 0,C 180,E1 -20848.263,E2 -20848.263} C_VEL
LIN {X 0,Y 213.821,Z 331.315,A -85,B 0,C 180,E1 -20852.604,E2 -20852.604} C_VEL
LIN {X 0,Y 213.847,Z 331.347,A -85,B 0,C 180,E1 -20856.954,E2 -20856.954} C_VEL
LIN {X 0,Y 213.938,Z 331.309,A -85,B 0,C 180,E1 -20862.804,E2 -20862.804} C_VEL
LIN {X 0,Y 213.946,Z 331.325,A -85,B 0,C 180,E1 -20866.707,E2 -20866.707} C_VEL
LIN {X 0,Y 214.136,Z 331.263,A -85,B 0,C 180,E1 -20870.556,E2 -20870.556} C_VEL
LIN {X 0,Y 214.095,Z 331.315,A -85,B 0,C 180,E1 -20874.349,E2 -20874.349} C_VEL
LIN {X 0,Y 214.439,Z 331.232,A -85,B 0,C 180,E1 -20878.123,E2 -20878.123} C_VEL
LIN {X 0,Y 214.541,Z 331.21,A -85,B 0,C 180,E1 -20880.001,E2 -20880.001} C_VEL
LIN {X 0,Y 214.44,Z 331.241,A -85,B 0,C 180,E1 -20881.879,E2 -20881.879} C_VEL
LIN {X 0,Y 214.194,Z 331.269,A -85,B 0,C 180,E1 -20887.543,E2 -20887.543} C_VEL
LIN {X 0,Y 213.995,Z 331.292,A -85,B 0,C 180,E1 -20891.366,E2 -20891.366} C_VEL
LIN {X 0,Y 213.927,Z 331.329,A -85,B 0,C 180,E1 -20895.238,E2 -20895.238} C_VEL
LIN {X 0,Y 213.831,Z 331.305,A -85,B 0,C 180,E1 -20899.189,E2 -20899.189} C_VEL
LIN {X 0,Y 213.808,Z 331.349,A -85,B 0,C 180,E1 -20903.233,E2 -20903.233} C_VEL
LIN {X 0,Y 213.828,Z 331.314,A -85,B 0,C 180,E1 -20907.451,E2 -20907.451} C_VEL
LIN {X 0,Y 213.766,Z 331.349,A -85,B 0,C 180,E1 -20911.739,E2 -20911.739} C_VEL
LIN {X 0,Y 213.743,Z 331.352,A -85,B 0,C 180,E1 -20916.29,E2 -20916.29} C_VEL
LIN {X 0,Y 213.704,Z 331.352,A -85,B 0,C 180,E1 -20921.128,E2 -20921.128} C_VEL
LIN {X 0,Y 213.737,Z 331.507,A -85,B 0,C 180,E1 -20925.575,E2 -20925.575} C_VEL
LIN {X 0,Y 215.233,Z 338.031,A -85,B 0,C 180,E1 -20930.116,E2 -20930.116} C_VEL
LIN {X 0,Y 215.549,Z 339.105,A -85,B 0,C 180,E1 -20930.564,E2 -20930.564} C_VEL
LIN {X 0,Y 217.756,Z 343.194,A -85,B 0,C 180,E1 -20931.248,E2 -20931.248} C_VEL
LIN {X 0,Y 224.649,Z 356.812,A -85,B 0,C 180,E1 -20933.169,E2 -20933.169} C_VEL
LIN {X 0,Y 231.897,Z 373.433,A -85,B 0,C 180,E1 -20935.106,E2 -20935.106} C_VEL
LIN {X 0,Y 232.774,Z 376.615,A -85,B 0,C 180,E1 -20935.372,E2 -20935.372} C_VEL
LIN {X 0,Y 236.032,Z 396.857,A -85,B 0,C 180,E1 -20936.636,E2 -20936.636} C_VEL
LIN {X 0,Y 234.088,Z 444.731,A -85,B 0,C 180,E1 -20938.084,E2 -20938.084} C_VEL
LIN {X 0,Y 233.151,Z 455.321,A -85,B 0,C 180,E1 -20938.586,E2 -20938.586} C_VEL
LIN {X 0,Y 232.686,Z 459.495,A -85,B 0,C 180,E1 -20938.822,E2 -20938.822} C_VEL
LIN {X 0,Y 231.333,Z 465.115,A -85,B 0,C 180,E1 -20939.122,E2 -20939.122} C_VEL
LIN {X 0,Y 227.356,Z 474.014,A -85,B 0,C 180,E1 -20939.569,E2 -20939.569} C_VEL
LIN {X 0,Y 223.154,Z 482.755,A -85,B 0,C 180,E1 -20940.193,E2 -20940.193} C_VEL
LIN {X 0,Y 221.452,Z 487.837,A -85,B 0,C 180,E1 -20940.771,E2 -20940.771} C_VEL
LIN {X 0,Y 218.779,Z 498.565,A -85,B 0,C 180,E1 -20942.499,E2 -20942.499} C_VEL
LIN {X 0,Y 216.639,Z 506.306,A -85,B 0,C 180,E1 -20944.027,E2 -20944.027} C_VEL
LIN {X 0,Y 213.919,Z 515.441,A -85,B 0,C 180,E1 -20946.269,E2 -20946.269} C_VEL
LIN {X 0,Y 211.944,Z 521.92,A -85,B 0,C 180,E1 -20948.2,E2 -20948.2} C_VEL
LIN {X 0,Y 210.039,Z 528.181,A -85,B 0,C 180,E1 -20950.452,E2 -20950.452} C_VEL
LIN {X 0,Y 208.649,Z 532.684,A -85,B 0,C 180,E1 -20952.354,E2 -20952.354} C_VEL
LIN {X 0,Y 206.808,Z 538.174,A -85,B 0,C 180,E1 -20955.234,E2 -20955.234} C_VEL
LIN {X 0,Y 205.581,Z 542.502,A -85,B 0,C 180,E1 -20958.164,E2 -20958.164} C_VEL
LIN {X 0,Y 205.054,Z 544.874,A -85,B 0,C 180,E1 -20960.133,E2 -20960.133} C_VEL
LIN {X 0,Y 204.628,Z 546.676,A -85,B 0,C 180,E1 -20962.104,E2 -20962.104} C_VEL
LIN {X 0,Y 204.339,Z 549.132,A -85,B 0,C 180,E1 -20966.056,E2 -20966.056} C_VEL
LIN {X 0,Y 204.332,Z 549.725,A -85,B 0,C 180,E1 -20968.029,E2 -20968.029} C_VEL
LIN {X 0,Y 204.438,Z 549.883,A -85,B 0,C 180,E1 -20970,E2 -20970} C_VEL
LIN {X 0,Y 204.331,Z 549.725,A -85,B 0,C 180,E1 -20971.971,E2 -20971.971} C_VEL
LIN {X 0,Y 204.299,Z 549.131,A -85,B 0,C 180,E1 -20973.945,E2 -20973.945} C_VEL
LIN {X 0,Y 204.614,Z 546.675,A -85,B 0,C 180,E1 -20977.897,E2 -20977.897} C_VEL
LIN {X 0,Y 205.284,Z 543.721,A -85,B 0,C 180,E1 -20980.853,E2 -20980.853} C_VEL
LIN {X 0,Y 206.314,Z 539.728,A -85,B 0,C 180,E1 -20983.795,E2 -20983.795} C_VEL
LIN {X 0,Y 207.951,Z 534.598,A -85,B 0,C 180,E1 -20986.694,E2 -20986.694} C_VEL
LIN {X 0,Y 209.635,Z 529.336,A -85,B 0,C 180,E1 -20989.078,E2 -20989.078} C_VEL
LIN {X 0,Y 211.732,Z 523.022,A -85,B 0,C 180,E1 -20991.415,E2 -20991.415} C_VEL
LIN {X 0,Y 213.442,Z 517.068,A -85,B 0,C 180,E1 -20993.273,E2 -20993.273} C_VEL
LIN {X 0,Y 215.503,Z 510.143,A -85,B 0,C 180,E1 -20995.084,E2 -20995.084} C_VEL
LIN {X 0,Y 217.86,Z 501.968,A -85,B 0,C 180,E1 -20996.848,E2 -20996.848} C_VEL
LIN {X 0,Y 220.074,Z 493.461,A -85,B 0,C 180,E1 -20998.36,E2 -20998.36} C_VEL
LIN {X 0,Y 222.121,Z 484.75,A -85,B 0,C 180,E1 -20999.628,E2 -20999.628} C_VEL
LIN {X 0,Y 224.059,Z 474.995,A -85,B 0,C 180,E1 -21000.774,E2 -21000.774} C_VEL
LIN {X 0,Y 225.56,Z 466.206,A -85,B 0,C 180,E1 -21001.59,E2 -21001.59} C_VEL
LIN {X 0,Y 227.01,Z 456.094,A -85,B 0,C 180,E1 -21002.292,E2 -21002.292} C_VEL
LIN {X 0,Y 228.043,Z 445.235,A -85,B 0,C 180,E1 -21002.827,E2 -21002.827} C_VEL
LIN {X 0,Y 230.07,Z 397.223,A -85,B 0,C 180,E1 -21004.326,E2 -21004.326} C_VEL
LIN {X 0,Y 226.729,Z 377.316,A -85,B 0,C 180,E1 -21005.656,E2 -21005.656} C_VEL
LIN {X 0,Y 220.724,Z 363.129,A -85,B 0,C 180,E1 -21007.339,E2 -21007.339} C_VEL
LIN {X 0,Y 213.262,Z 347.825,A -85,B 0,C 180,E1 -21009.523,E2 -21009.523} C_VEL
LIN {X 0,Y 209.82,Z 342.085,A -85,B 0,C 180,E1 -21010.55,E2 -21010.55} C_VEL
LIN {X 0,Y 208.11,Z 338.44,A -85,B 0,C 180,E1 -21011.23,E2 -21011.23} C_VEL
LIN {X 0,Y 206.683,Z 332.39,A -85,B 0,C 180,E1 -21015.566,E2 -21015.566} C_VEL
LIN {X 0,Y 206.652,Z 332.225,A -85,B 0,C 180,E1 -21019.745,E2 -21019.745} C_VEL
LIN {X 0,Y 206.698,Z 332.215,A -85,B 0,C 180,E1 -21024.687,E2 -21024.687} C_VEL
LIN {X 0,Y 206.706,Z 332.238,A -85,B 0,C 180,E1 -21029.335,E2 -21029.335} C_VEL
LIN {X 0,Y 206.728,Z 332.197,A -85,B 0,C 180,E1 -21033.77,E2 -21033.77} C_VEL
LIN {X 0,Y 206.737,Z 332.226,A -85,B 0,C 180,E1 -21038.04,E2 -21038.04} C_VEL
LIN {X 0,Y 206.869,Z 332.172,A -85,B 0,C 180,E1 -21042.195,E2 -21042.195} C_VEL
LIN {X 0,Y 206.889,Z 332.21,A -85,B 0,C 180,E1 -21046.243,E2 -21046.243} C_VEL
LIN {X 0,Y 207.096,Z 332.137,A -85,B 0,C 180,E1 -21050.23,E2 -21050.23} C_VEL
LIN {X 0,Y 207.057,Z 332.185,A -85,B 0,C 180,E1 -21054.155,E2 -21054.155} C_VEL
LIN {X 0,Y 207.377,Z 332.121,A -85,B 0,C 180,E1 -21058.057,E2 -21058.057} C_VEL
LIN {X 0,Y 207.506,Z 332.085,A -85,B 0,C 180,E1 -21059.999,E2 -21059.999} C_VEL
LIN {X 0,Y 207.376,Z 332.112,A -85,B 0,C 180,E1 -21061.941,E2 -21061.941} C_VEL
LIN {X 0,Y 207.135,Z 332.152,A -85,B 0,C 180,E1 -21067.799,E2 -21067.799} C_VEL
LIN {X 0,Y 206.918,Z 332.172,A -85,B 0,C 180,E1 -21071.758,E2 -21071.758} C_VEL
LIN {X 0,Y 206.861,Z 332.212,A -85,B 0,C 180,E1 -21075.77,E2 -21075.77} C_VEL
LIN {X 0,Y 206.778,Z 332.187,A -85,B 0,C 180,E1 -21079.868,E2 -21079.868} C_VEL
LIN {X 0,Y 206.758,Z 332.229,A -85,B 0,C 180,E1 -21084.072,E2 -21084.072} C_VEL
LIN {X 0,Y 206.732,Z 332.202,A -85,B 0,C 180,E1 -21088.419,E2 -21088.419} C_VEL
LIN {X 0,Y 206.7,Z 332.22,A -85,B 0,C 180,E1 -21092.956,E2 -21092.956} C_VEL
LIN {X 0,Y 206.72,Z 332.238,A -85,B 0,C 180,E1 -21097.73,E2 -21097.73} C_VEL
LIN {X 0,Y 206.718,Z 332.216,A -85,B 0,C 180,E1 -21101.588,E2 -21101.588} C_VEL
LIN {X 0,Y 206.656,Z 332.195,A -85,B 0,C 180,E1 -21105.574,E2 -21105.574} C_VEL
LIN {X 0,Y 206.691,Z 332.42,A -85,B 0,C 180,E1 -21108.334,E2 -21108.334} C_VEL
LIN {X 0,Y 207.003,Z 333.605,A -85,B 0,C 180,E1 -21108.766,E2 -21108.766} C_VEL
LIN {X 0,Y 208.676,Z 336.305,A -85,B 0,C 180,E1 -21109.31,E2 -21109.31} C_VEL
LIN {X 0,Y 209.701,Z 337.641,A -85,B 0,C 180,E1 -21109.611,E2 -21109.611} C_VEL
LIN {X 0,Y 218.237,Z 351.203,A -85,B 0,C 180,E1 -21112.062,E2 -21112.062} C_VEL
LIN {X 0,Y 227.045,Z 367.399,A -85,B 0,C 180,E1 -21114.407,E2 -21114.407} C_VEL
LIN {X 0,Y 235.96,Z 385.284,A -85,B 0,C 180,E1 -21116.596,E2 -21116.596} C_VEL
LIN {X 0,Y 243.812,Z 397.708,A -85,B 0,C 180,E1 -21118.236,E2 -21118.236} C_VEL
LIN {X 0,Y 251.806,Z 408.345,A -85,B 0,C 180,E1 -21119.71,E2 -21119.71} C_VEL
LIN {X 0,Y 264.71,Z 422.738,A -85,B 0,C 180,E1 -21121.776,E2 -21121.776} C_VEL
LIN {X 0,Y 276.809,Z 434.387,A -85,B 0,C 180,E1 -21123.503,E2 -21123.503} C_VEL
LIN {X 0,Y 287.555,Z 443.647,A -85,B 0,C 180,E1 -21125.036,E2 -21125.036} C_VEL
LIN {X 0,Y 298.601,Z 452.536,A -85,B 0,C 180,E1 -21126.621,E2 -21126.621} C_VEL
LIN {X 0,Y 307.016,Z 459.053,A -85,B 0,C 180,E1 -21127.984,E2 -21127.984} C_VEL
LIN {X 0,Y 315.178,Z 464.931,A -85,B 0,C 180,E1 -21129.475,E2 -21129.475} C_VEL
LIN {X 0,Y 321.835,Z 469.958,A -85,B 0,C 180,E1 -21130.88,E2 -21130.88} C_VEL
LIN {X 0,Y 329.435,Z 475.084,A -85,B 0,C 180,E1 -21132.623,E2 -21132.623} C_VEL
LIN {X 0,Y 335.757,Z 479.707,A -85,B 0,C 180,E1 -21134.333,E2 -21134.333} C_VEL
LIN {X 0,Y 340.752,Z 482.834,A -85,B 0,C 180,E1 -21135.78,E2 -21135.78} C_VEL
LIN {X 0,Y 345.687,Z 485.787,A -85,B 0,C 180,E1 -21137.383,E2 -21137.383} C_VEL
LIN {X 0,Y 350.428,Z 489.314,A -85,B 0,C 180,E1 -21139.328,E2 -21139.328} C_VEL
LIN {X 0,Y 355.179,Z 492.307,A -85,B 0,C 180,E1 -21141.629,E2 -21141.629} C_VEL
LIN {X 0,Y 357.979,Z 493.723,A -85,B 0,C 180,E1 -21143.235,E2 -21143.235} C_VEL
LIN {X 0,Y 359.998,Z 494.59,A -85,B 0,C 180,E1 -21144.639,E2 -21144.639} C_VEL
LIN {X 0,Y 362.146,Z 495.324,A -85,B 0,C 180,E1 -21146.662,E2 -21146.662} C_VEL
LIN {X 0,Y 362.822,Z 495.704,A -85,B 0,C 180,E1 -21147.78,E2 -21147.78} C_VEL
LIN {X 0,Y 363.199,Z 495.961,A -85,B 0,C 180,E1 -21148.891,E2 -21148.891} C_VEL
LIN {X 0,Y 363.42,Z 495.904,A -85,B 0,C 180,E1 -21150,E2 -21150} C_VEL
LIN {X 0,Y 363.238,Z 495.89,A -85,B 0,C 180,E1 -21151.109,E2 -21151.109} C_VEL
LIN {X 0,Y 362.833,Z 495.66,A -85,B 0,C 180,E1 -21152.22,E2 -21152.22} C_VEL
LIN {X 0,Y 362.118,Z 495.325,A -85,B 0,C 180,E1 -21153.338,E2 -21153.338} C_VEL
LIN {X 0,Y 359.99,Z 494.595,A -85,B 0,C 180,E1 -21155.349,E2 -21155.349} C_VEL
LIN {X 0,Y 357.958,Z 493.72,A -85,B 0,C 180,E1 -21156.765,E2 -21156.765} C_VEL
LIN {X 0,Y 355.193,Z 492.281,A -85,B 0,C 180,E1 -21158.387,E2 -21158.387} C_VEL
LIN {X 0,Y 350.423,Z 489.302,A -85,B 0,C 180,E1 -21160.667,E2 -21160.667} C_VEL
LIN {X 0,Y 345.676,Z 485.779,A -85,B 0,C 180,E1 -21162.609,E2 -21162.609} C_VEL
LIN {X 0,Y 340.288,Z 482.598,A -85,B 0,C 180,E1 -21164.349,E2 -21164.349} C_VEL
LIN {X 0,Y 333.1,Z 477.785,A -85,B 0,C 180,E1 -21166.407,E2 -21166.407} C_VEL
LIN {X 0,Y 327.614,Z 473.77,A -85,B 0,C 180,E1 -21167.827,E2 -21167.827} C_VEL
LIN {X 0,Y 320.441,Z 468.936,A -85,B 0,C 180,E1 -21169.426,E2 -21169.426} C_VEL
LIN {X 0,Y 313.61,Z 463.755,A -85,B 0,C 180,E1 -21170.833,E2 -21170.833} C_VEL
LIN {X 0,Y 305.641,Z 457.992,A -85,B 0,C 180,E1 -21172.255,E2 -21172.255} C_VEL
LIN {X 0,Y 296.89,Z 451.248,A -85,B 0,C 180,E1 -21173.627,E2 -21173.627} C_VEL
LIN {X 0,Y 281.729,Z 438.833,A -85,B 0,C 180,E1 -21175.792,E2 -21175.792} C_VEL
LIN {X 0,Y 269.476,Z 427.485,A -85,B 0,C 180,E1 -21177.537,E2 -21177.537} C_VEL
LIN {X 0,Y 255.815,Z 413.133,A -85,B 0,C 180,E1 -21179.611,E2 -21179.611} C_VEL
LIN {X 0,Y 246.227,Z 401.144,A -85,B 0,C 180,E1 -21181.299,E2 -21181.299} C_VEL
LIN {X 0,Y 237.792,Z 388.405,A -85,B 0,C 180,E1 -21183.001,E2 -21183.001} C_VEL
LIN {X 0,Y 230.372,Z 374.384,A -85,B 0,C 180,E1 -21184.738,E2 -21184.738} C_VEL
LIN {X 0,Y 224.373,Z 362.369,A -85,B 0,C 180,E1 -21186.282,E2 -21186.282} C_VEL
LIN {X 0,Y 216.441,Z 348.146,A -85,B 0,C 180,E1 -21188.44,E2 -21188.44} C_VEL
LIN {X 0,Y 210.877,Z 339.674,A -85,B 0,C 180,E1 -21190.027,E2 -21190.027} C_VEL
LIN {X 0,Y 209.036,Z 336.66,A -85,B 0,C 180,E1 -21190.589,E2 -21190.589} C_VEL
LIN {X 0,Y 207.201,Z 334.104,A -85,B 0,C 180,E1 -21191.151,E2 -21191.151} C_VEL
LIN {X 0,Y 206.759,Z 332.772,A -85,B 0,C 180,E1 -21191.454,E2 -21191.454} C_VEL
LIN {X 0,Y 206.629,Z 332.22,A -85,B 0,C 180,E1 -21192.133,E2 -21192.133} C_VEL
LIN {X 0,Y 206.711,Z 332.232,A -85,B 0,C 180,E1 -21197.159,E2 -21197.159} C_VEL
LIN {X 0,Y 206.755,Z 332.226,A -85,B 0,C 180,E1 -21201.425,E2 -21201.425} C_VEL
LIN {X 0,Y 206.726,Z 332.209,A -85,B 0,C 180,E1 -21204.695,E2 -21204.695} C_VEL
LIN {X 0,Y 206.702,Z 332.237,A -85,B 0,C 180,E1 -21209.337,E2 -21209.337} C_VEL
LIN {X 0,Y 206.726,Z 332.203,A -85,B 0,C 180,E1 -21213.773,E2 -21213.773} C_VEL
LIN {X 0,Y 206.752,Z 332.217,A -85,B 0,C 180,E1 -21218.044,E2 -21218.044} C_VEL
LIN {X 0,Y 206.868,Z 332.181,A -85,B 0,C 180,E1 -21222.197,E2 -21222.197} C_VEL
LIN {X 0,Y 206.889,Z 332.209,A -85,B 0,C 180,E1 -21226.245,E2 -21226.245} C_VEL
LIN {X 0,Y 207.095,Z 332.138,A -85,B 0,C 180,E1 -21230.232,E2 -21230.232} C_VEL
LIN {X 0,Y 207.056,Z 332.191,A -85,B 0,C 180,E1 -21234.157,E2 -21234.157} C_VEL
LIN {X 0,Y 207.376,Z 332.112,A -85,B 0,C 180,E1 -21238.059,E2 -21238.059} C_VEL
LIN {X 0,Y 207.506,Z 332.085,A -85,B 0,C 180,E1 -21240.001,E2 -21240.001} C_VEL
LIN {X 0,Y 207.377,Z 332.121,A -85,B 0,C 180,E1 -21241.943,E2 -21241.943} C_VEL
LIN {X 0,Y 207.136,Z 332.143,A -85,B 0,C 180,E1 -21247.801,E2 -21247.801} C_VEL
LIN {X 0,Y 206.92,Z 332.179,A -85,B 0,C 180,E1 -21251.76,E2 -21251.76} C_VEL
LIN {X 0,Y 206.861,Z 332.2,A -85,B 0,C 180,E1 -21255.772,E2 -21255.772} C_VEL
LIN {X 0,Y 206.759,Z 332.19,A -85,B 0,C 180,E1 -21259.873,E2 -21259.873} C_VEL
LIN {X 0,Y 206.744,Z 332.221,A -85,B 0,C 180,E1 -21264.076,E2 -21264.076} C_VEL
LIN {X 0,Y 206.735,Z 332.206,A -85,B 0,C 180,E1 -21268.421,E2 -21268.421} C_VEL
LIN {X 0,Y 206.697,Z 332.213,A -85,B 0,C 180,E1 -21272.959,E2 -21272.959} C_VEL
LIN {X 0,Y 206.674,Z 332.239,A -85,B 0,C 180,E1 -21277.742,E2 -21277.742} C_VEL
LIN {X 0,Y 206.636,Z 332.237,A -85,B 0,C 180,E1 -21281.562,E2 -21281.562} C_VEL
LIN {X 0,Y 206.683,Z 332.391,A -85,B 0,C 180,E1 -21284.434,E2 -21284.434} C_VEL
LIN {X 0,Y 208.048,Z 338.373,A -85,B 0,C 180,E1 -21288.725,E2 -21288.725} C_VEL
LIN {X 0,Y 209.408,Z 341.456,A -85,B 0,C 180,E1 -21289.326,E2 -21289.326} C_VEL
LIN {X 0,Y 211.315,Z 344.613,A -85,B 0,C 180,E1 -21289.903,E2 -21289.903} C_VEL
LIN {X 0,Y 215.923,Z 353.167,A -85,B 0,C 180,E1 -21291.276,E2 -21291.276} C_VEL
LIN {X 0,Y 222.197,Z 366.341,A -85,B 0,C 180,E1 -21293.075,E2 -21293.075} C_VEL
LIN {X 0,Y 227.003,Z 378.26,A -85,B 0,C 180,E1 -21294.429,E2 -21294.429} C_VEL
LIN {X 0,Y 230.042,Z 397.364,A -85,B 0,C 180,E1 -21295.674,E2 -21295.674} C_VEL
LIN {X 0,Y 228.053,Z 445.265,A -85,B 0,C 180,E1 -21297.173,E2 -21297.173} C_VEL
LIN {X 0,Y 227.023,Z 456.086,A -85,B 0,C 180,E1 -21297.709,E2 -21297.709} C_VEL
LIN {X 0,Y 225.417,Z 467.494,A -85,B 0,C 180,E1 -21298.519,E2 -21298.519} C_VEL
LIN {X 0,Y 223.146,Z 479.854,A -85,B 0,C 180,E1 -21299.741,E2 -21299.741} C_VEL
LIN {X 0,Y 221.452,Z 487.837,A -85,B 0,C 180,E1 -21300.771,E2 -21300.771} C_VEL
LIN {X 0,Y 219.684,Z 492.92,A -85,B 0,C 180,E1 -21301.411,E2 -21301.411} C_VEL
LIN {X 0,Y 215.042,Z 500.794,A -85,B 0,C 180,E1 -21302.439,E2 -21302.439} C_VEL
LIN {X 0,Y 210.279,Z 508.138,A -85,B 0,C 180,E1 -21303.696,E2 -21303.696} C_VEL
LIN {X 0,Y 208.352,Z 512.388,A -85,B 0,C 180,E1 -21304.687,E2 -21304.687} C_VEL
LIN {X 0,Y 205.395,Z 521.586,A -85,B 0,C 180,E1 -21307.414,E2 -21307.414} C_VEL
LIN {X 0,Y 203.355,Z 527.987,A -85,B 0,C 180,E1 -21309.782,E2 -21309.782} C_VEL
LIN {X 0,Y 201.86,Z 532.489,A -85,B 0,C 180,E1 -21311.739,E2 -21311.739} C_VEL
LIN {X 0,Y 199.909,Z 537.978,A -85,B 0,C 180,E1 -21314.712,E2 -21314.712} C_VEL
LIN {X 0,Y 198.605,Z 542.307,A -85,B 0,C 180,E1 -21317.742,E2 -21317.742} C_VEL
LIN {X 0,Y 198.023,Z 544.679,A -85,B 0,C 180,E1 -21319.779,E2 -21319.779} C_VEL
LIN {X 0,Y 197.581,Z 546.482,A -85,B 0,C 180,E1 -21321.82,E2 -21321.82} C_VEL
LIN {X 0,Y 197.247,Z 548.988,A -85,B 0,C 180,E1 -21326.086,E2 -21326.086} C_VEL
LIN {X 0,Y 197.241,Z 549.531,A -85,B 0,C 180,E1 -21327.958,E2 -21327.958} C_VEL
LIN {X 0,Y 197.339,Z 549.689,A -85,B 0,C 180,E1 -21330,E2 -21330} C_VEL
LIN {X 0,Y 197.237,Z 549.531,A -85,B 0,C 180,E1 -21332.042,E2 -21332.042} C_VEL
LIN {X 0,Y 197.21,Z 548.937,A -85,B 0,C 180,E1 -21334.087,E2 -21334.087} C_VEL
LIN {X 0,Y 197.57,Z 546.481,A -85,B 0,C 180,E1 -21338.18,E2 -21338.18} C_VEL
LIN {X 0,Y 198.274,Z 543.526,A -85,B 0,C 180,E1 -21341.242,E2 -21341.242} C_VEL
LIN {X 0,Y 199.387,Z 539.533,A -85,B 0,C 180,E1 -21344.284,E2 -21344.284} C_VEL
LIN {X 0,Y 201.139,Z 534.403,A -85,B 0,C 180,E1 -21347.277,E2 -21347.277} C_VEL
LIN {X 0,Y 202.919,Z 529.141,A -85,B 0,C 180,E1 -21349.735,E2 -21349.735} C_VEL
LIN {X 0,Y 204.666,Z 524.203,A -85,B 0,C 180,E1 -21351.662,E2 -21351.662} C_VEL
LIN {X 0,Y 206.915,Z 516.873,A -85,B 0,C 180,E1 -21354.053,E2 -21354.053} C_VEL
LIN {X 0,Y 209.068,Z 509.948,A -85,B 0,C 180,E1 -21355.912,E2 -21355.912} C_VEL
LIN {X 0,Y 211.51,Z 501.773,A -85,B 0,C 180,E1 -21357.722,E2 -21357.722} C_VEL
LIN {X 0,Y 213.855,Z 493.268,A -85,B 0,C 180,E1 -21359.264,E2 -21359.264} C_VEL
LIN {X 0,Y 215.978,Z 484.556,A -85,B 0,C 180,E1 -21360.559,E2 -21360.559} C_VEL
LIN {X 0,Y 217.989,Z 474.801,A -85,B 0,C 180,E1 -21361.729,E2 -21361.729} C_VEL
LIN {X 0,Y 219.555,Z 466.012,A -85,B 0,C 180,E1 -21362.558,E2 -21362.558} C_VEL
LIN {X 0,Y 221.128,Z 455.432,A -85,B 0,C 180,E1 -21363.297,E2 -21363.297} C_VEL
LIN {X 0,Y 222.058,Z 445.835,A -85,B 0,C 180,E1 -21363.789,E2 -21363.789} C_VEL
LIN {X 0,Y 223.521,Z 416.401,A -85,B 0,C 180,E1 -21364.736,E2 -21364.736} C_VEL
LIN {X 0,Y 224.202,Z 398.424,A -85,B 0,C 180,E1 -21365.303,E2 -21365.303} C_VEL
LIN {X 0,Y 221.221,Z 380.182,A -85,B 0,C 180,E1 -21366.565,E2 -21366.565} C_VEL
LIN {X 0,Y 215.613,Z 366.79,A -85,B 0,C 180,E1 -21368.223,E2 -21368.223} C_VEL
LIN {X 0,Y 208.571,Z 352.155,A -85,B 0,C 180,E1 -21370.396,E2 -21370.396} C_VEL
LIN {X 0,Y 202.544,Z 341.767,A -85,B 0,C 180,E1 -21372.337,E2 -21372.337} C_VEL
LIN {X 0,Y 200.805,Z 338.203,A -85,B 0,C 180,E1 -21373.08,E2 -21373.08} C_VEL
LIN {X 0,Y 200.05,Z 335.031,A -85,B 0,C 180,E1 -21375.361,E2 -21375.361} C_VEL
LIN {X 0,Y 199.6,Z 333.131,A -85,B 0,C 180,E1 -21377.052,E2 -21377.052} C_VEL
LIN {X 0,Y 199.6,Z 333.104,A -85,B 0,C 180,E1 -21380.77,E2 -21380.77} C_VEL
LIN {X 0,Y 199.613,Z 333.104,A -85,B 0,C 180,E1 -21384.073,E2 -21384.073} C_VEL
LIN {X 0,Y 199.692,Z 333.098,A -85,B 0,C 180,E1 -21388.134,E2 -21388.134} C_VEL
LIN {X 0,Y 199.682,Z 333.074,A -85,B 0,C 180,E1 -21392.77,E2 -21392.77} C_VEL
LIN {X 0,Y 199.712,Z 333.107,A -85,B 0,C 180,E1 -21397.225,E2 -21397.225} C_VEL
LIN {X 0,Y 199.793,Z 333.051,A -85,B 0,C 180,E1 -21401.758,E2 -21401.758} C_VEL
LIN {X 0,Y 199.83,Z 333.091,A -85,B 0,C 180,E1 -21405.747,E2 -21405.747} C_VEL
LIN {X 0,Y 200.019,Z 333.019,A -85,B 0,C 180,E1 -21409.88,E2 -21409.88} C_VEL
LIN {X 0,Y 200.019,Z 333.059,A -85,B 0,C 180,E1 -21413.948,E2 -21413.948} C_VEL
LIN {X 0,Y 200.316,Z 333,A -85,B 0,C 180,E1 -21417.988,E2 -21417.988} C_VEL
LIN {X 0,Y 200.471,Z 332.961,A -85,B 0,C 180,E1 -21419.999,E2 -21419.999} C_VEL
LIN {X 0,Y 200.021,Z 333.062,A -85,B 0,C 180,E1 -21424.029,E2 -21424.029} C_VEL
LIN {X 0,Y 200.084,Z 333.025,A -85,B 0,C 180,E1 -21428.076,E2 -21428.076} C_VEL
LIN {X 0,Y 199.869,Z 333.056,A -85,B 0,C 180,E1 -21432.179,E2 -21432.179} C_VEL
LIN {X 0,Y 199.799,Z 333.083,A -85,B 0,C 180,E1 -21436.343,E2 -21436.343} C_VEL
LIN {X 0,Y 199.694,Z 333.074,A -85,B 0,C 180,E1 -21440.605,E2 -21440.605} C_VEL
LIN {X 0,Y 199.667,Z 333.098,A -85,B 0,C 180,E1 -21444.984,E2 -21444.984} C_VEL
LIN {X 0,Y 199.66,Z 333.095,A -85,B 0,C 180,E1 -21449.523,E2 -21449.523} C_VEL
LIN {X 0,Y 199.652,Z 333.105,A -85,B 0,C 180,E1 -21452.349,E2 -21452.349} C_VEL
LIN {X 0,Y 199.648,Z 333.106,A -85,B 0,C 180,E1 -21456.756,E2 -21456.756} C_VEL
LIN {X 0,Y 199.673,Z 333.097,A -85,B 0,C 180,E1 -21459.311,E2 -21459.311} C_VEL
LIN {X 0,Y 199.657,Z 333.102,A -85,B 0,C 180,E1 -21462.338,E2 -21462.338} C_VEL
LIN {X 0,Y 199.631,Z 333.308,A -85,B 0,C 180,E1 -21466.519,E2 -21466.519} C_VEL
LIN {X 0,Y 199.843,Z 334.265,A -85,B 0,C 180,E1 -21466.944,E2 -21466.944} C_VEL
LIN {X 0,Y 201.438,Z 337.046,A -85,B 0,C 180,E1 -21467.538,E2 -21467.538} C_VEL
LIN {X 0,Y 202.685,Z 338.491,A -85,B 0,C 180,E1 -21467.929,E2 -21467.929} C_VEL
LIN {X 0,Y 205.031,Z 341.959,A -85,B 0,C 180,E1 -21468.681,E2 -21468.681} C_VEL
LIN {X 0,Y 213.819,Z 356.067,A -85,B 0,C 180,E1 -21471.332,E2 -21471.332} C_VEL
LIN {X 0,Y 222.005,Z 371.333,A -85,B 0,C 180,E1 -21473.619,E2 -21473.619} C_VEL
LIN {X 0,Y 231.113,Z 389.775,A -85,B 0,C 180,E1 -21475.959,E2 -21475.959} C_VEL
LIN {X 0,Y 239.045,Z 402.429,A -85,B 0,C 180,E1 -21477.686,E2 -21477.686} C_VEL
LIN {X 0,Y 247.059,Z 413.19,A -85,B 0,C 180,E1 -21479.22,E2 -21479.22} C_VEL
LIN {X 0,Y 260.346,Z 428.108,A -85,B 0,C 180,E1 -21481.421,E2 -21481.421} C_VEL
LIN {X 0,Y 271.683,Z 439.195,A -85,B 0,C 180,E1 -21483.182,E2 -21483.182} C_VEL
LIN {X 0,Y 282.582,Z 448.738,A -85,B 0,C 180,E1 -21484.883,E2 -21484.883} C_VEL
LIN {X 0,Y 294.044,Z 457.982,A -85,B 0,C 180,E1 -21486.648,E2 -21486.648} C_VEL
LIN {X 0,Y 301.613,Z 463.837,A -85,B 0,C 180,E1 -21487.852,E2 -21487.852} C_VEL
LIN {X 0,Y 310.754,Z 470.467,A -85,B 0,C 180,E1 -21489.504,E2 -21489.504} C_VEL
LIN {X 0,Y 316.464,Z 474.834,A -85,B 0,C 180,E1 -21490.702,E2 -21490.702} C_VEL
LIN {X 0,Y 324.309,Z 480.116,A -85,B 0,C 180,E1 -21492.458,E2 -21492.458} C_VEL
LIN {X 0,Y 329.842,Z 484.212,A -85,B 0,C 180,E1 -21493.92,E2 -21493.92} C_VEL
LIN {X 0,Y 335.135,Z 487.71,A -85,B 0,C 180,E1 -21495.425,E2 -21495.425} C_VEL
LIN {X 0,Y 341.104,Z 491.238,A -85,B 0,C 180,E1 -21497.308,E2 -21497.308} C_VEL
LIN {X 0,Y 344.196,Z 493.576,A -85,B 0,C 180,E1 -21498.545,E2 -21498.545} C_VEL
LIN {X 0,Y 346.391,Z 495.111,A -85,B 0,C 180,E1 -21499.479,E2 -21499.479} C_VEL
LIN {X 0,Y 349.069,Z 496.875,A -85,B 0,C 180,E1 -21500.731,E2 -21500.731} C_VEL
LIN {X 0,Y 351.437,Z 498.232,A -85,B 0,C 180,E1 -21501.953,E2 -21501.953} C_VEL
LIN {X 0,Y 353.797,Z 499.416,A -85,B 0,C 180,E1 -21503.319,E2 -21503.319} C_VEL
LIN {X 0,Y 355.267,Z 500.09,A -85,B 0,C 180,E1 -21504.324,E2 -21504.324} C_VEL
LIN {X 0,Y 356.697,Z 500.68,A -85,B 0,C 180,E1 -21505.48,E2 -21505.48} C_VEL
LIN {X 0,Y 357.866,Z 500.996,A -85,B 0,C 180,E1 -21506.622,E2 -21506.622} C_VEL
LIN {X 0,Y 358.658,Z 501.441,A -85,B 0,C 180,E1 -21507.928,E2 -21507.928} C_VEL
LIN {X 0,Y 359.181,Z 501.573,A -85,B 0,C 180,E1 -21510,E2 -21510} C_VEL
LIN {X 0,Y 358.655,Z 501.396,A -85,B 0,C 180,E1 -21512.062,E2 -21512.062} C_VEL
LIN {X 0,Y 357.833,Z 500.998,A -85,B 0,C 180,E1 -21513.378,E2 -21513.378} C_VEL
LIN {X 0,Y 356.693,Z 500.639,A -85,B 0,C 180,E1 -21514.52,E2 -21514.52} C_VEL
LIN {X 0,Y 355.244,Z 500.071,A -85,B 0,C 180,E1 -21515.677,E2 -21515.677} C_VEL
LIN {X 0,Y 353.471,Z 499.285,A -85,B 0,C 180,E1 -21516.851,E2 -21516.851} C_VEL
LIN {X 0,Y 351.415,Z 498.228,A -85,B 0,C 180,E1 -21518.047,E2 -21518.047} C_VEL
LIN {X 0,Y 348.976,Z 496.758,A -85,B 0,C 180,E1 -21519.322,E2 -21519.322} C_VEL
LIN {X 0,Y 346.374,Z 495.1,A -85,B 0,C 180,E1 -21520.522,E2 -21520.522} C_VEL
LIN {X 0,Y 343.304,Z 492.933,A -85,B 0,C 180,E1 -21521.813,E2 -21521.813} C_VEL
LIN {X 0,Y 339.381,Z 490.201,A -85,B 0,C 180,E1 -21523.276,E2 -21523.276} C_VEL
LIN {X 0,Y 334.372,Z 487.191,A -85,B 0,C 180,E1 -21524.797,E2 -21524.797} C_VEL
LIN {X 0,Y 328.01,Z 482.83,A -85,B 0,C 180,E1 -21526.584,E2 -21526.584} C_VEL
LIN {X 0,Y 321.721,Z 478.407,A -85,B 0,C 180,E1 -21528.148,E2 -21528.148} C_VEL
LIN {X 0,Y 313.835,Z 472.881,A -85,B 0,C 180,E1 -21529.859,E2 -21529.859} C_VEL
LIN {X 0,Y 308.493,Z 468.818,A -85,B 0,C 180,E1 -21530.927,E2 -21530.927} C_VEL
LIN {X 0,Y 300.211,Z 462.732,A -85,B 0,C 180,E1 -21532.379,E2 -21532.379} C_VEL
LIN {X 0,Y 290.251,Z 455.08,A -85,B 0,C 180,E1 -21533.93,E2 -21533.93} C_VEL
LIN {X 0,Y 275.778,Z 442.955,A -85,B 0,C 180,E1 -21536.168,E2 -21536.168} C_VEL
LIN {X 0,Y 264.857,Z 432.657,A -85,B 0,C 180,E1 -21537.88,E2 -21537.88} C_VEL
LIN {X 0,Y 251.394,Z 418.4,A -85,B 0,C 180,E1 -21540.02,E2 -21540.02} C_VEL
LIN {X 0,Y 241.436,Z 405.879,A -85,B 0,C 180,E1 -21541.835,E2 -21541.835} C_VEL
LIN {X 0,Y 232.761,Z 392.625,A -85,B 0,C 180,E1 -21543.662,E2 -21543.662} C_VEL
LIN {X 0,Y 225.259,Z 378.262,A -85,B 0,C 180,E1 -21545.502,E2 -21545.502} C_VEL
LIN {X 0,Y 219.384,Z 366.313,A -85,B 0,C 180,E1 -21547.092,E2 -21547.092} C_VEL
LIN {X 0,Y 211.837,Z 352.726,A -85,B 0,C 180,E1 -21549.245,E2 -21549.245} C_VEL
LIN {X 0,Y 204.604,Z 341.474,A -85,B 0,C 180,E1 -21551.447,E2 -21551.447} C_VEL
LIN {X 0,Y 201.959,Z 337.56,A -85,B 0,C 180,E1 -21552.302,E2 -21552.302} C_VEL
LIN {X 0,Y 200.149,Z 335.065,A -85,B 0,C 180,E1 -21552.904,E2 -21552.904} C_VEL
LIN {X 0,Y 199.694,Z 333.628,A -85,B 0,C 180,E1 -21553.256,E2 -21553.256} C_VEL
LIN {X 0,Y 199.613,Z 333.195,A -85,B 0,C 180,E1 -21553.638,E2 -21553.638} C_VEL
LIN {X 0,Y 199.661,Z 333.098,A -85,B 0,C 180,E1 -21558.028,E2 -21558.028} C_VEL
LIN {X 0,Y 199.675,Z 333.098,A -85,B 0,C 180,E1 -21560.743,E2 -21560.743} C_VEL
LIN {X 0,Y 199.627,Z 333.09,A -85,B 0,C 180,E1 -21565.718,E2 -21565.718} C_VEL
LIN {X 0,Y 199.691,Z 333.108,A -85,B 0,C 180,E1 -21568.137,E2 -21568.137} C_VEL
LIN {X 0,Y 199.68,Z 333.075,A -85,B 0,C 180,E1 -21572.772,E2 -21572.772} C_VEL
LIN {X 0,Y 199.733,Z 333.103,A -85,B 0,C 180,E1 -21577.23,E2 -21577.23} C_VEL
LIN {X 0,Y 199.791,Z 333.057,A -85,B 0,C 180,E1 -21581.759,E2 -21581.759} C_VEL
LIN {X 0,Y 199.83,Z 333.093,A -85,B 0,C 180,E1 -21585.749,E2 -21585.749} C_VEL
LIN {X 0,Y 200.018,Z 333.019,A -85,B 0,C 180,E1 -21589.883,E2 -21589.883} C_VEL
LIN {X 0,Y 200.017,Z 333.067,A -85,B 0,C 180,E1 -21593.95,E2 -21593.95} C_VEL
LIN {X 0,Y 200.315,Z 332.991,A -85,B 0,C 180,E1 -21597.991,E2 -21597.991} C_VEL
LIN {X 0,Y 200.471,Z 332.961,A -85,B 0,C 180,E1 -21600.001,E2 -21600.001} C_VEL
LIN {X 0,Y 200.023,Z 333.068,A -85,B 0,C 180,E1 -21604.031,E2 -21604.031} C_VEL
LIN {X 0,Y 200.085,Z 333.017,A -85,B 0,C 180,E1 -21608.078,E2 -21608.078} C_VEL
LIN {X 0,Y 199.87,Z 333.063,A -85,B 0,C 180,E1 -21612.181,E2 -21612.181} C_VEL
LIN {X 0,Y 199.799,Z 333.068,A -85,B 0,C 180,E1 -21616.345,E2 -21616.345} C_VEL
LIN {X 0,Y 199.679,Z 333.081,A -85,B 0,C 180,E1 -21620.609,E2 -21620.609} C_VEL
LIN {X 0,Y 199.662,Z 333.088,A -85,B 0,C 180,E1 -21624.987,E2 -21624.987} C_VEL
LIN {X 0,Y 199.663,Z 333.104,A -85,B 0,C 180,E1 -21629.525,E2 -21629.525} C_VEL
LIN {X 0,Y 199.67,Z 333.094,A -85,B 0,C 180,E1 -21632.357,E2 -21632.357} C_VEL
LIN {X 0,Y 199.62,Z 333.117,A -85,B 0,C 180,E1 -21636.765,E2 -21636.765} C_VEL
LIN {X 0,Y 199.598,Z 333.104,A -85,B 0,C 180,E1 -21639.332,E2 -21639.332} C_VEL
LIN {X 0,Y 199.643,Z 333.331,A -85,B 0,C 180,E1 -21643.263,E2 -21643.263} C_VEL
LIN {X 0,Y 200.704,Z 337.802,A -85,B 0,C 180,E1 -21646.72,E2 -21646.72} C_VEL
LIN {X 0,Y 201.014,Z 338.854,A -85,B 0,C 180,E1 -21647.088,E2 -21647.088} C_VEL
LIN {X 0,Y 203.376,Z 342.974,A -85,B 0,C 180,E1 -21647.931,E2 -21647.931} C_VEL
LIN {X 0,Y 210.731,Z 356.314,A -85,B 0,C 180,E1 -21650.279,E2 -21650.279} C_VEL
LIN {X 0,Y 217.93,Z 371.934,A -85,B 0,C 180,E1 -21652.461,E2 -21652.461} C_VEL
LIN {X 0,Y 221.374,Z 380.511,A -85,B 0,C 180,E1 -21653.477,E2 -21653.477} C_VEL
LIN {X 0,Y 224.193,Z 398.554,A -85,B 0,C 180,E1 -21654.7,E2 -21654.7} C_VEL
LIN {X 0,Y 222.144,Z 444.806,A -85,B 0,C 180,E1 -21656.169,E2 -21656.169} C_VEL
LIN {X 0,Y 221.108,Z 455.416,A -85,B 0,C 180,E1 -21656.698,E2 -21656.698} C_VEL
LIN {X 0,Y 219.613,Z 466.014,A -85,B 0,C 180,E1 -21657.451,E2 -21657.451} C_VEL
LIN {X 0,Y 217.665,Z 476.817,A -85,B 0,C 180,E1 -21658.49,E2 -21658.49} C_VEL
LIN {X 0,Y 214.91,Z 489.215,A -85,B 0,C 180,E1 -21660.086,E2 -21660.086} C_VEL
LIN {X 0,Y 212.175,Z 499.505,A -85,B 0,C 180,E1 -21661.836,E2 -21661.836} C_VEL
LIN {X 0,Y 209.673,Z 508.03,A -85,B 0,C 180,E1 -21663.633,E2 -21663.633} C_VEL
LIN {X 0,Y 208.352,Z 512.388,A -85,B 0,C 180,E1 -21664.687,E2 -21664.687} C_VEL
LIN {X 0,Y 206.447,Z 516.477,A -85,B 0,C 180,E1 -21665.749,E2 -21665.749} C_VEL
LIN {X 0,Y 201.725,Z 522.777,A -85,B 0,C 180,E1 -21667.454,E2 -21667.454} C_VEL
LIN {X 0,Y 197.079,Z 528.469,A -85,B 0,C 180,E1 -21669.371,E2 -21669.371} C_VEL
LIN {X 0,Y 195.339,Z 531.603,A -85,B 0,C 180,E1 -21670.744,E2 -21670.744} C_VEL
LIN {X 0,Y 193.039,Z 537.784,A -85,B 0,C 180,E1 -21674.154,E2 -21674.154} C_VEL
LIN {X 0,Y 191.651,Z 542.113,A -85,B 0,C 180,E1 -21677.29,E2 -21677.29} C_VEL
LIN {X 0,Y 191.011,Z 544.484,A -85,B 0,C 180,E1 -21679.399,E2 -21679.399} C_VEL
LIN {X 0,Y 190.533,Z 546.287,A -85,B 0,C 180,E1 -21681.516,E2 -21681.516} C_VEL
LIN {X 0,Y 190.166,Z 548.744,A -85,B 0,C 180,E1 -21685.761,E2 -21685.761} C_VEL
LIN {X 0,Y 190.152,Z 549.337,A -85,B 0,C 180,E1 -21687.882,E2 -21687.882} C_VEL
LIN {X 0,Y 190.243,Z 549.495,A -85,B 0,C 180,E1 -21690,E2 -21690} C_VEL
LIN {X 0,Y 190.12,Z 548.942,A -85,B 0,C 180,E1 -21693.529,E2 -21693.529} C_VEL
LIN {X 0,Y 190.234,Z 547.679,A -85,B 0,C 180,E1 -21696.363,E2 -21696.363} C_VEL
LIN {X 0,Y 190.524,Z 546.287,A -85,B 0,C 180,E1 -21698.485,E2 -21698.485} C_VEL
LIN {X 0,Y 191.285,Z 543.331,A -85,B 0,C 180,E1 -21701.658,E2 -21701.658} C_VEL
LIN {X 0,Y 192.475,Z 539.338,A -85,B 0,C 180,E1 -21704.809,E2 -21704.809} C_VEL
LIN {X 0,Y 194.35,Z 534.209,A -85,B 0,C 180,E1 -21707.901,E2 -21707.901} C_VEL
LIN {X 0,Y 196.239,Z 528.947,A -85,B 0,C 180,E1 -21710.437,E2 -21710.437} C_VEL
LIN {X 0,Y 198.153,Z 523.646,A -85,B 0,C 180,E1 -21712.557,E2 -21712.557} C_VEL
LIN {X 0,Y 200.419,Z 516.678,A -85,B 0,C 180,E1 -21714.884,E2 -21714.884} C_VEL
LIN {X 0,Y 202.7,Z 509.754,A -85,B 0,C 180,E1 -21716.79,E2 -21716.79} C_VEL
LIN {X 0,Y 205.244,Z 501.579,A -85,B 0,C 180,E1 -21718.645,E2 -21718.645} C_VEL
LIN {X 0,Y 207.683,Z 493.074,A -85,B 0,C 180,E1 -21720.222,E2 -21720.222} C_VEL
LIN {X 0,Y 209.895,Z 484.362,A -85,B 0,C 180,E1 -21721.545,E2 -21721.545} C_VEL
LIN {X 0,Y 211.961,Z 474.607,A -85,B 0,C 180,E1 -21722.742,E2 -21722.742} C_VEL
LIN {X 0,Y 213.619,Z 465.819,A -85,B 0,C 180,E1 -21723.581,E2 -21723.581} C_VEL
LIN {X 0,Y 215.197,Z 455.476,A -85,B 0,C 180,E1 -21724.322,E2 -21724.322} C_VEL
LIN {X 0,Y 216.213,Z 445.37,A -85,B 0,C 180,E1 -21724.846,E2 -21724.846} C_VEL
LIN {X 0,Y 217.992,Z 409.671,A -85,B 0,C 180,E1 -21726.01,E2 -21726.01} C_VEL
LIN {X 0,Y 218.35,Z 399.008,A -85,B 0,C 180,E1 -21726.367,E2 -21726.367} C_VEL
LIN {X 0,Y 215.626,Z 382.494,A -85,B 0,C 180,E1 -21727.573,E2 -21727.573} C_VEL
LIN {X 0,Y 209.484,Z 367.904,A -85,B 0,C 180,E1 -21729.498,E2 -21729.498} C_VEL
LIN {X 0,Y 203.425,Z 355.589,A -85,B 0,C 180,E1 -21731.474,E2 -21731.474} C_VEL
LIN {X 0,Y 198.031,Z 346.108,A -85,B 0,C 180,E1 -21733.319,E2 -21733.319} C_VEL
LIN {X 0,Y 195.509,Z 341.824,A -85,B 0,C 180,E1 -21734.229,E2 -21734.229} C_VEL
LIN {X 0,Y 193.559,Z 337.989,A -85,B 0,C 180,E1 -21735.107,E2 -21735.107} C_VEL
LIN {X 0,Y 192.536,Z 334.087,A -85,B 0,C 180,E1 -21738.217,E2 -21738.217} C_VEL
LIN {X 0,Y 192.584,Z 333.989,A -85,B 0,C 180,E1 -21743.401,E2 -21743.401} C_VEL
LIN {X 0,Y 192.607,Z 333.967,A -85,B 0,C 180,E1 -21747.058,E2 -21747.058} C_VEL
LIN {X 0,Y 192.659,Z 333.956,A -85,B 0,C 180,E1 -21751.69,E2 -21751.69} C_VEL
LIN {X 0,Y 192.683,Z 333.977,A -85,B 0,C 180,E1 -21756.344,E2 -21756.344} C_VEL
LIN {X 0,Y 192.728,Z 333.93,A -85,B 0,C 180,E1 -21761.458,E2 -21761.458} C_VEL
LIN {X 0,Y 192.758,Z 333.968,A -85,B 0,C 180,E1 -21765.212,E2 -21765.212} C_VEL
LIN {X 0,Y 192.942,Z 333.901,A -85,B 0,C 180,E1 -21769.565,E2 -21769.565} C_VEL
LIN {X 0,Y 192.981,Z 333.931,A -85,B 0,C 180,E1 -21773.727,E2 -21773.727} C_VEL
LIN {X 0,Y 193.258,Z 333.879,A -85,B 0,C 180,E1 -21777.915,E2 -21777.915} C_VEL
LIN {X 0,Y 193.436,Z 333.836,A -85,B 0,C 180,E1 -21779.999,E2 -21779.999} C_VEL
LIN {X 0,Y 192.967,Z 333.942,A -85,B 0,C 180,E1 -21784.176,E2 -21784.176} C_VEL
LIN {X 0,Y 193.031,Z 333.898,A -85,B 0,C 180,E1 -21788.373,E2 -21788.373} C_VEL
LIN {X 0,Y 192.797,Z 333.943,A -85,B 0,C 180,E1 -21792.632,E2 -21792.632} C_VEL
LIN {X 0,Y 192.752,Z 333.948,A -85,B 0,C 180,E1 -21796.958,E2 -21796.958} C_VEL
LIN {X 0,Y 192.631,Z 333.963,A -85,B 0,C 180,E1 -21801.397,E2 -21801.397} C_VEL
LIN {X 0,Y 192.659,Z 333.982,A -85,B 0,C 180,E1 -21804.224,E2 -21804.224} C_VEL
LIN {X 0,Y 192.639,Z 333.96,A -85,B 0,C 180,E1 -21808.888,E2 -21808.888} C_VEL
LIN {X 0,Y 192.593,Z 333.973,A -85,B 0,C 180,E1 -21813.185,E2 -21813.185} C_VEL
LIN {X 0,Y 192.595,Z 333.992,A -85,B 0,C 180,E1 -21818.34,E2 -21818.34} C_VEL
LIN {X 0,Y 192.593,Z 333.993,A -85,B 0,C 180,E1 -21823.129,E2 -21823.129} C_VEL
LIN {X 0,Y 192.633,Z 334.236,A -85,B 0,C 180,E1 -21824.633,E2 -21824.633} C_VEL
LIN {X 0,Y 192.92,Z 335.382,A -85,B 0,C 180,E1 -21825.053,E2 -21825.053} C_VEL
LIN {X 0,Y 194.52,Z 338.082,A -85,B 0,C 180,E1 -21825.683,E2 -21825.683} C_VEL
LIN {X 0,Y 195.716,Z 339.358,A -85,B 0,C 180,E1 -21826.09,E2 -21826.09} C_VEL
LIN {X 0,Y 197.961,Z 342.8,A -85,B 0,C 180,E1 -21826.885,E2 -21826.885} C_VEL
LIN {X 0,Y 203.729,Z 351.553,A -85,B 0,C 180,E1 -21828.8,E2 -21828.8} C_VEL
LIN {X 0,Y 209.876,Z 361.746,A -85,B 0,C 180,E1 -21830.707,E2 -21830.707} C_VEL
LIN {X 0,Y 217.584,Z 376.442,A -85,B 0,C 180,E1 -21832.959,E2 -21832.959} C_VEL
LIN {X 0,Y 225.595,Z 392.941,A -85,B 0,C 180,E1 -21835.121,E2 -21835.121} C_VEL
LIN {X 0,Y 233.634,Z 406.175,A -85,B 0,C 180,E1 -21836.971,E2 -21836.971} C_VEL
LIN {X 0,Y 242.036,Z 417.668,A -85,B 0,C 180,E1 -21838.657,E2 -21838.657} C_VEL
LIN {X 0,Y 254.666,Z 432.127,A -85,B 0,C 180,E1 -21840.88,E2 -21840.88} C_VEL
LIN {X 0,Y 265.058,Z 442.673,A -85,B 0,C 180,E1 -21842.652,E2 -21842.652} C_VEL
LIN {X 0,Y 276.275,Z 452.794,A -85,B 0,C 180,E1 -21844.56,E2 -21844.56} C_VEL
LIN {X 0,Y 290.374,Z 464.008,A -85,B 0,C 180,E1 -21846.883,E2 -21846.883} C_VEL
LIN {X 0,Y 300.183,Z 471.542,A -85,B 0,C 180,E1 -21848.533,E2 -21848.533} C_VEL
LIN {X 0,Y 307.959,Z 477.22,A -85,B 0,C 180,E1 -21849.982,E2 -21849.982} C_VEL
LIN {X 0,Y 314.998,Z 482.348,A -85,B 0,C 180,E1 -21851.482,E2 -21851.482} C_VEL
LIN {X 0,Y 321.427,Z 486.755,A -85,B 0,C 180,E1 -21852.992,E2 -21852.992} C_VEL
LIN {X 0,Y 327.814,Z 491.337,A -85,B 0,C 180,E1 -21854.74,E2 -21854.74} C_VEL
LIN {X 0,Y 334.146,Z 495.21,A -85,B 0,C 180,E1 -21856.623,E2 -21856.623} C_VEL
LIN {X 0,Y 338.078,Z 497.805,A -85,B 0,C 180,E1 -21858.002,E2 -21858.002} C_VEL
LIN {X 0,Y 342.61,Z 501.03,A -85,B 0,C 180,E1 -21859.937,E2 -21859.937} C_VEL
LIN {X 0,Y 347.432,Z 503.929,A -85,B 0,C 180,E1 -21862.384,E2 -21862.384} C_VEL
LIN {X 0,Y 350.409,Z 505.336,A -85,B 0,C 180,E1 -21864.245,E2 -21864.245} C_VEL
LIN {X 0,Y 352.332,Z 506.12,A -85,B 0,C 180,E1 -21865.821,E2 -21865.821} C_VEL
LIN {X 0,Y 353.137,Z 506.335,A -85,B 0,C 180,E1 -21866.577,E2 -21866.577} C_VEL
LIN {X 0,Y 353.875,Z 506.729,A -85,B 0,C 180,E1 -21867.724,E2 -21867.724} C_VEL
LIN {X 0,Y 354.31,Z 506.959,A -85,B 0,C 180,E1 -21868.863,E2 -21868.863} C_VEL
LIN {X 0,Y 354.549,Z 506.925,A -85,B 0,C 180,E1 -21870,E2 -21870} C_VEL
LIN {X 0,Y 354.35,Z 506.899,A -85,B 0,C 180,E1 -21871.136,E2 -21871.136} C_VEL
LIN {X 0,Y 353.904,Z 506.671,A -85,B 0,C 180,E1 -21872.276,E2 -21872.276} C_VEL
LIN {X 0,Y 352.345,Z 506.102,A -85,B 0,C 180,E1 -21874.208,E2 -21874.208} C_VEL
LIN {X 0,Y 350.374,Z 505.324,A -85,B 0,C 180,E1 -21875.756,E2 -21875.756} C_VEL
LIN {X 0,Y 347.437,Z 503.953,A -85,B 0,C 180,E1 -21877.622,E2 -21877.622} C_VEL
LIN {X 0,Y 342.613,Z 501.014,A -85,B 0,C 180,E1 -21880.066,E2 -21880.066} C_VEL
LIN {X 0,Y 338.027,Z 497.787,A -85,B 0,C 180,E1 -21882,E2 -21882} C_VEL
LIN {X 0,Y 334.157,Z 495.227,A -85,B 0,C 180,E1 -21883.376,E2 -21883.376} C_VEL
LIN {X 0,Y 327.823,Z 491.286,A -85,B 0,C 180,E1 -21885.266,E2 -21885.266} C_VEL
LIN {X 0,Y 322.77,Z 487.736,A -85,B 0,C 180,E1 -21886.656,E2 -21886.656} C_VEL
LIN {X 0,Y 316.925,Z 483.635,A -85,B 0,C 180,E1 -21888.086,E2 -21888.086} C_VEL
LIN {X 0,Y 309.69,Z 478.571,A -85,B 0,C 180,E1 -21889.651,E2 -21889.651} C_VEL
LIN {X 0,Y 304.34,Z 474.488,A -85,B 0,C 180,E1 -21890.734,E2 -21890.734} C_VEL
LIN {X 0,Y 296.004,Z 468.397,A -85,B 0,C 180,E1 -21892.187,E2 -21892.187} C_VEL
LIN {X 0,Y 281.449,Z 457.05,A -85,B 0,C 180,E1 -21894.582,E2 -21894.582} C_VEL
LIN {X 0,Y 269.633,Z 446.867,A -85,B 0,C 180,E1 -21896.576,E2 -21896.576} C_VEL
LIN {X 0,Y 259.631,Z 437.242,A -85,B 0,C 180,E1 -21898.288,E2 -21898.288} C_VEL
LIN {X 0,Y 248.301,Z 425.137,A -85,B 0,C 180,E1 -21900.214,E2 -21900.214} C_VEL
LIN {X 0,Y 237.455,Z 411.726,A -85,B 0,C 180,E1 -21902.232,E2 -21902.232} C_VEL
LIN {X 0,Y 228.215,Z 397.617,A -85,B 0,C 180,E1 -21904.244,E2 -21904.244} C_VEL
LIN {X 0,Y 220.774,Z 383.357,A -85,B 0,C 180,E1 -21906.141,E2 -21906.141} C_VEL
LIN {X 0,Y 214.24,Z 369.888,A -85,B 0,C 180,E1 -21907.997,E2 -21907.997} C_VEL
LIN {X 0,Y 207.362,Z 357.356,A -85,B 0,C 180,E1 -21910.063,E2 -21910.063} C_VEL
LIN {X 0,Y 200.319,Z 346.294,A -85,B 0,C 180,E1 -21912.316,E2 -21912.316} C_VEL
LIN {X 0,Y 197.815,Z 342.643,A -85,B 0,C 180,E1 -21913.163,E2 -21913.163} C_VEL
LIN {X 0,Y 195.624,Z 339.189,A -85,B 0,C 180,E1 -21913.944,E2 -21913.944} C_VEL
LIN {X 0,Y 193.424,Z 336.552,A -85,B 0,C 180,E1 -21914.715,E2 -21914.715} C_VEL
LIN {X 0,Y 192.712,Z 334.665,A -85,B 0,C 180,E1 -21915.138,E2 -21915.138} C_VEL
LIN {X 0,Y 192.592,Z 334.047,A -85,B 0,C 180,E1 -21915.606,E2 -21915.606} C_VEL
LIN {X 0,Y 192.585,Z 333.974,A -85,B 0,C 180,E1 -21920.026,E2 -21920.026} C_VEL
LIN {X 0,Y 192.597,Z 333.97,A -85,B 0,C 180,E1 -21924.28,E2 -21924.28} C_VEL
LIN {X 0,Y 192.594,Z 333.995,A -85,B 0,C 180,E1 -21929.279,E2 -21929.279} C_VEL
LIN {X 0,Y 192.655,Z 333.953,A -85,B 0,C 180,E1 -21931.692,E2 -21931.692} C_VEL
LIN {X 0,Y 192.701,Z 333.982,A -85,B 0,C 180,E1 -21936.349,E2 -21936.349} C_VEL
LIN {X 0,Y 192.727,Z 333.935,A -85,B 0,C 180,E1 -21941.459,E2 -21941.459} C_VEL
LIN {X 0,Y 192.758,Z 333.976,A -85,B 0,C 180,E1 -21945.215,E2 -21945.215} C_VEL
LIN {X 0,Y 192.941,Z 333.9,A -85,B 0,C 180,E1 -21949.568,E2 -21949.568} C_VEL
LIN {X 0,Y 192.98,Z 333.94,A -85,B 0,C 180,E1 -21953.729,E2 -21953.729} C_VEL
LIN {X 0,Y 193.257,Z 333.87,A -85,B 0,C 180,E1 -21957.917,E2 -21957.917} C_VEL
LIN {X 0,Y 193.436,Z 333.836,A -85,B 0,C 180,E1 -21960.001,E2 -21960.001} C_VEL
LIN {X 0,Y 192.969,Z 333.947,A -85,B 0,C 180,E1 -21964.178,E2 -21964.178} C_VEL
LIN {X 0,Y 193.032,Z 333.891,A -85,B 0,C 180,E1 -21968.375,E2 -21968.375} C_VEL
LIN {X 0,Y 192.798,Z 333.952,A -85,B 0,C 180,E1 -21972.635,E2 -21972.635} C_VEL
LIN {X 0,Y 192.753,Z 333.936,A -85,B 0,C 180,E1 -21976.96,E2 -21976.96} C_VEL
LIN {X 0,Y 192.614,Z 333.973,A -85,B 0,C 180,E1 -21981.401,E2 -21981.401} C_VEL
LIN {X 0,Y 192.645,Z 333.973,A -85,B 0,C 180,E1 -21984.214,E2 -21984.214} C_VEL
LIN {X 0,Y 192.643,Z 333.966,A -85,B 0,C 180,E1 -21988.89,E2 -21988.89} C_VEL
LIN {X 0,Y 192.595,Z 333.966,A -85,B 0,C 180,E1 -21993.188,E2 -21993.188} C_VEL
LIN {X 0,Y 192.544,Z 333.989,A -85,B 0,C 180,E1 -21998.355,E2 -21998.355} C_VEL
LIN {X 0,Y 192.537,Z 334.108,A -85,B 0,C 180,E1 -22001.787,E2 -22001.787} C_VEL
LIN {X 0,Y 193.572,Z 337.966,A -85,B 0,C 180,E1 -22004.889,E2 -22004.889} C_VEL
LIN {X 0,Y 195.661,Z 342.041,A -85,B 0,C 180,E1 -22005.825,E2 -22005.825} C_VEL
LIN {X 0,Y 197.468,Z 345.193,A -85,B 0,C 180,E1 -22006.483,E2 -22006.483} C_VEL
LIN {X 0,Y 202.685,Z 354.298,A -85,B 0,C 180,E1 -22008.282,E2 -22008.282} C_VEL
LIN {X 0,Y 208.162,Z 365.049,A -85,B 0,C 180,E1 -22010.078,E2 -22010.078} C_VEL
LIN {X 0,Y 214.549,Z 379.729,A -85,B 0,C 180,E1 -22012.092,E2 -22012.092} C_VEL
LIN {X 0,Y 215.999,Z 383.823,A -85,B 0,C 180,E1 -22012.557,E2 -22012.557} C_VEL
LIN {X 0,Y 218.425,Z 400.411,A -85,B 0,C 180,E1 -22013.703,E2 -22013.703} C_VEL
LIN {X 0,Y 216.286,Z 444.397,A -85,B 0,C 180,E1 -22015.11,E2 -22015.11} C_VEL
LIN {X 0,Y 215.271,Z 454.786,A -85,B 0,C 180,E1 -22015.636,E2 -22015.636} C_VEL
LIN {X 0,Y 213.89,Z 464.534,A -85,B 0,C 180,E1 -22016.326,E2 -22016.326} C_VEL
LIN {X 0,Y 212.246,Z 473.603,A -85,B 0,C 180,E1 -22017.166,E2 -22017.166} C_VEL
LIN {X 0,Y 210.254,Z 482.731,A -85,B 0,C 180,E1 -22018.234,E2 -22018.234} C_VEL
LIN {X 0,Y 208.019,Z 491.722,A -85,B 0,C 180,E1 -22019.551,E2 -22019.551} C_VEL
LIN {X 0,Y 205.577,Z 500.445,A -85,B 0,C 180,E1 -22021.127,E2 -22021.127} C_VEL
LIN {X 0,Y 203.317,Z 507.836,A -85,B 0,C 180,E1 -22022.742,E2 -22022.742} C_VEL
LIN {X 0,Y 200.966,Z 515.052,A -85,B 0,C 180,E1 -22024.635,E2 -22024.635} C_VEL
LIN {X 0,Y 198.87,Z 521.252,A -85,B 0,C 180,E1 -22026.574,E2 -22026.574} C_VEL
LIN {X 0,Y 196.704,Z 527.793,A -85,B 0,C 180,E1 -22029.067,E2 -22029.067} C_VEL
LIN {X 0,Y 195.339,Z 531.603,A -85,B 0,C 180,E1 -22030.744,E2 -22030.744} C_VEL
LIN {X 0,Y 193.66,Z 534.489,A -85,B 0,C 180,E1 -22032.183,E2 -22032.183} C_VEL
LIN {X 0,Y 191.17,Z 537.155,A -85,B 0,C 180,E1 -22033.594,E2 -22033.594} C_VEL
LIN {X 0,Y 185.274,Z 542.232,A -85,B 0,C 180,E1 -22037.094,E2 -22037.094} C_VEL
LIN {X 0,Y 184.046,Z 544.076,A -85,B 0,C 180,E1 -22038.787,E2 -22038.787} C_VEL
LIN {X 0,Y 183.504,Z 546.093,A -85,B 0,C 180,E1 -22041.188,E2 -22041.188} C_VEL
LIN {X 0,Y 183.08,Z 548.55,A -85,B 0,C 180,E1 -22045.597,E2 -22045.597} C_VEL
LIN {X 0,Y 183.05,Z 549.143,A -85,B 0,C 180,E1 -22047.8,E2 -22047.8} C_VEL
LIN {X 0,Y 183.15,Z 549.302,A -85,B 0,C 180,E1 -22050,E2 -22050} C_VEL
LIN {X 0,Y 183.035,Z 548.847,A -85,B 0,C 180,E1 -22053.301,E2 -22053.301} C_VEL
LIN {X 0,Y 183.181,Z 547.485,A -85,B 0,C 180,E1 -22056.609,E2 -22056.609} C_VEL
LIN {X 0,Y 183.498,Z 546.093,A -85,B 0,C 180,E1 -22058.812,E2 -22058.812} C_VEL
LIN {X 0,Y 184.318,Z 543.137,A -85,B 0,C 180,E1 -22062.105,E2 -22062.105} C_VEL
LIN {X 0,Y 185.582,Z 539.143,A -85,B 0,C 180,E1 -22065.372,E2 -22065.372} C_VEL
LIN {X 0,Y 187.587,Z 534.014,A -85,B 0,C 180,E1 -22068.569,E2 -22068.569} C_VEL
LIN {X 0,Y 189.597,Z 528.753,A -85,B 0,C 180,E1 -22071.186,E2 -22071.186} C_VEL
LIN {X 0,Y 191.375,Z 524.059,A -85,B 0,C 180,E1 -22073.149,E2 -22073.149} C_VEL
LIN {X 0,Y 193.429,Z 518.11,A -85,B 0,C 180,E1 -22075.272,E2 -22075.272} C_VEL
LIN {X 0,Y 196.384,Z 509.56,A -85,B 0,C 180,E1 -22077.725,E2 -22077.725} C_VEL
LIN {X 0,Y 199.026,Z 501.385,A -85,B 0,C 180,E1 -22079.627,E2 -22079.627} C_VEL
LIN {X 0,Y 201.573,Z 492.879,A -85,B 0,C 180,E1 -22081.239,E2 -22081.239} C_VEL
LIN {X 0,Y 203.879,Z 484.169,A -85,B 0,C 180,E1 -22082.589,E2 -22082.589} C_VEL
LIN {X 0,Y 206.018,Z 474.413,A -85,B 0,C 180,E1 -22083.812,E2 -22083.812} C_VEL
LIN {X 0,Y 208.001,Z 464.339,A -85,B 0,C 180,E1 -22084.762,E2 -22084.762} C_VEL
LIN {X 0,Y 209.485,Z 454.209,A -85,B 0,C 180,E1 -22085.486,E2 -22085.486} C_VEL
LIN {X 0,Y 210.504,Z 443.963,A -85,B 0,C 180,E1 -22086.002,E2 -22086.002} C_VEL
LIN {X 0,Y 212.632,Z 400.158,A -85,B 0,C 180,E1 -22087.454,E2 -22087.454} C_VEL
LIN {X 0,Y 210.232,Z 385.317,A -85,B 0,C 180,E1 -22088.584,E2 -22088.584} C_VEL
LIN {X 0,Y 204.475,Z 371.471,A -85,B 0,C 180,E1 -22090.496,E2 -22090.496} C_VEL
LIN {X 0,Y 198.544,Z 359.269,A -85,B 0,C 180,E1 -22092.546,E2 -22092.546} C_VEL
LIN {X 0,Y 191.726,Z 347.147,A -85,B 0,C 180,E1 -22095.056,E2 -22095.056} C_VEL
LIN {X 0,Y 188.921,Z 342.436,A -85,B 0,C 180,E1 -22096.161,E2 -22096.161} C_VEL
LIN {X 0,Y 186.384,Z 338.262,A -85,B 0,C 180,E1 -22097.254,E2 -22097.254} C_VEL
LIN {X 0,Y 186.021,Z 337.152,A -85,B 0,C 180,E1 -22097.774,E2 -22097.774} C_VEL
LIN {X 0,Y 185.465,Z 334.887,A -85,B 0,C 180,E1 -22099.893,E2 -22099.893} C_VEL
LIN {X 0,Y 185.503,Z 334.879,A -85,B 0,C 180,E1 -22102.711,E2 -22102.711} C_VEL
LIN {X 0,Y 185.541,Z 334.856,A -85,B 0,C 180,E1 -22107.973,E2 -22107.973} C_VEL
LIN {X 0,Y 185.579,Z 334.853,A -85,B 0,C 180,E1 -22110.575,E2 -22110.575} C_VEL
LIN {X 0,Y 185.579,Z 334.845,A -85,B 0,C 180,E1 -22115.38,E2 -22115.38} C_VEL
LIN {X 0,Y 185.671,Z 334.808,A -85,B 0,C 180,E1 -22121.134,E2 -22121.134} C_VEL
LIN {X 0,Y 185.69,Z 334.84,A -85,B 0,C 180,E1 -22124.636,E2 -22124.636} C_VEL
LIN {X 0,Y 185.886,Z 334.78,A -85,B 0,C 180,E1 -22129.417,E2 -22129.417} C_VEL
LIN {X 0,Y 185.944,Z 334.8,A -85,B 0,C 180,E1 -22133.488,E2 -22133.488} C_VEL
LIN {X 0,Y 186.202,Z 334.758,A -85,B 0,C 180,E1 -22137.836,E2 -22137.836} C_VEL
LIN {X 0,Y 186.4,Z 334.712,A -85,B 0,C 180,E1 -22139.999,E2 -22139.999} C_VEL
LIN {X 0,Y 185.914,Z 334.822,A -85,B 0,C 180,E1 -22144.335,E2 -22144.335} C_VEL
LIN {X 0,Y 185.978,Z 334.772,A -85,B 0,C 180,E1 -22148.693,E2 -22148.693} C_VEL
LIN {X 0,Y 185.724,Z 334.832,A -85,B 0,C 180,E1 -22153.122,E2 -22153.122} C_VEL
LIN {X 0,Y 185.685,Z 334.818,A -85,B 0,C 180,E1 -22157.624,E2 -22157.624} C_VEL
LIN {X 0,Y 185.591,Z 334.855,A -85,B 0,C 180,E1 -22162.251,E2 -22162.251} C_VEL
LIN {X 0,Y 185.555,Z 334.834,A -85,B 0,C 180,E1 -22167.032,E2 -22167.032} C_VEL
LIN {X 0,Y 185.573,Z 334.847,A -85,B 0,C 180,E1 -22169.493,E2 -22169.493} C_VEL
LIN {X 0,Y 185.515,Z 334.847,A -85,B 0,C 180,E1 -22174.627,E2 -22174.627} C_VEL
LIN {X 0,Y 185.563,Z 334.868,A -85,B 0,C 180,E1 -22177.313,E2 -22177.313} C_VEL
LIN {X 0,Y 185.524,Z 334.946,A -85,B 0,C 180,E1 -22182.223,E2 -22182.223} C_VEL
LIN {X 0,Y 185.727,Z 335.856,A -85,B 0,C 180,E1 -22182.777,E2 -22182.777} C_VEL
LIN {X 0,Y 187.372,Z 338.809,A -85,B 0,C 180,E1 -22183.533,E2 -22183.533} C_VEL
LIN {X 0,Y 188.912,Z 340.404,A -85,B 0,C 180,E1 -22184.111,E2 -22184.111} C_VEL
LIN {X 0,Y 190.994,Z 343.696,A -85,B 0,C 180,E1 -22184.928,E2 -22184.928} C_VEL
LIN {X 0,Y 192.229,Z 345.424,A -85,B 0,C 180,E1 -22185.388,E2 -22185.388} C_VEL
LIN {X 0,Y 197.988,Z 354.014,A -85,B 0,C 180,E1 -22187.438,E2 -22187.438} C_VEL
LIN {X 0,Y 205.176,Z 365.92,A -85,B 0,C 180,E1 -22189.805,E2 -22189.805} C_VEL
LIN {X 0,Y 212.938,Z 381.049,A -85,B 0,C 180,E1 -22192.196,E2 -22192.196} C_VEL
LIN {X 0,Y 221.143,Z 398.116,A -85,B 0,C 180,E1 -22194.51,E2 -22194.51} C_VEL
LIN {X 0,Y 229.369,Z 411.565,A -85,B 0,C 180,E1 -22196.469,E2 -22196.469} C_VEL
LIN {X 0,Y 237.517,Z 422.738,A -85,B 0,C 180,E1 -22198.163,E2 -22198.163} C_VEL
LIN {X 0,Y 248.841,Z 435.935,A -85,B 0,C 180,E1 -22200.279,E2 -22200.279} C_VEL
LIN {X 0,Y 260.684,Z 448.206,A -85,B 0,C 180,E1 -22202.515,E2 -22202.515} C_VEL
LIN {X 0,Y 272.195,Z 458.624,A -85,B 0,C 180,E1 -22204.645,E2 -22204.645} C_VEL
LIN {X 0,Y 286.092,Z 469.593,A -85,B 0,C 180,E1 -22207.101,E2 -22207.101} C_VEL
LIN {X 0,Y 298.918,Z 479.174,A -85,B 0,C 180,E1 -22209.35,E2 -22209.35} C_VEL
LIN {X 0,Y 305.409,Z 484.066,A -85,B 0,C 180,E1 -22210.642,E2 -22210.642} C_VEL
LIN {X 0,Y 313.346,Z 489.537,A -85,B 0,C 180,E1 -22212.372,E2 -22212.372} C_VEL
LIN {X 0,Y 318.531,Z 493.332,A -85,B 0,C 180,E1 -22213.689,E2 -22213.689} C_VEL
LIN {X 0,Y 325.252,Z 497.875,A -85,B 0,C 180,E1 -22215.56,E2 -22215.56} C_VEL
LIN {X 0,Y 331.233,Z 501.487,A -85,B 0,C 180,E1 -22217.421,E2 -22217.421} C_VEL
LIN {X 0,Y 336.078,Z 504.965,A -85,B 0,C 180,E1 -22219.371,E2 -22219.371} C_VEL
LIN {X 0,Y 338.428,Z 506.562,A -85,B 0,C 180,E1 -22220.437,E2 -22220.437} C_VEL
LIN {X 0,Y 340.969,Z 508.107,A -85,B 0,C 180,E1 -22221.704,E2 -22221.704} C_VEL
LIN {X 0,Y 343.234,Z 509.3,A -85,B 0,C 180,E1 -22222.943,E2 -22222.943} C_VEL
LIN {X 0,Y 345.85,Z 510.54,A -85,B 0,C 180,E1 -22224.692,E2 -22224.692} C_VEL
LIN {X 0,Y 347.981,Z 511.292,A -85,B 0,C 180,E1 -22226.526,E2 -22226.526} C_VEL
LIN {X 0,Y 348.778,Z 511.67,A -85,B 0,C 180,E1 -22227.69,E2 -22227.69} C_VEL
LIN {X 0,Y 349.236,Z 511.904,A -85,B 0,C 180,E1 -22228.847,E2 -22228.847} C_VEL
LIN {X 0,Y 349.478,Z 511.895,A -85,B 0,C 180,E1 -22230,E2 -22230} C_VEL
LIN {X 0,Y 349.273,Z 511.855,A -85,B 0,C 180,E1 -22231.153,E2 -22231.153} C_VEL
LIN {X 0,Y 348.793,Z 511.63,A -85,B 0,C 180,E1 -22232.31,E2 -22232.31} C_VEL
LIN {X 0,Y 347.963,Z 511.272,A -85,B 0,C 180,E1 -22233.474,E2 -22233.474} C_VEL
LIN {X 0,Y 345.86,Z 510.547,A -85,B 0,C 180,E1 -22235.325,E2 -22235.325} C_VEL
LIN {X 0,Y 343.188,Z 509.302,A -85,B 0,C 180,E1 -22237.058,E2 -22237.058} C_VEL
LIN {X 0,Y 340.925,Z 508.063,A -85,B 0,C 180,E1 -22238.318,E2 -22238.318} C_VEL
LIN {X 0,Y 338.446,Z 506.52,A -85,B 0,C 180,E1 -22239.562,E2 -22239.562} C_VEL
LIN {X 0,Y 334.466,Z 503.83,A -85,B 0,C 180,E1 -22241.321,E2 -22241.321} C_VEL
LIN {X 0,Y 331.237,Z 501.512,A -85,B 0,C 180,E1 -22242.582,E2 -22242.582} C_VEL
LIN {X 0,Y 325.276,Z 497.857,A -85,B 0,C 180,E1 -22244.439,E2 -22244.439} C_VEL
LIN {X 0,Y 318.539,Z 493.286,A -85,B 0,C 180,E1 -22246.316,E2 -22246.316} C_VEL
LIN {X 0,Y 313.296,Z 489.561,A -85,B 0,C 180,E1 -22247.636,E2 -22247.636} C_VEL
LIN {X 0,Y 305.41,Z 484.056,A -85,B 0,C 180,E1 -22249.358,E2 -22249.358} C_VEL
LIN {X 0,Y 298.881,Z 479.148,A -85,B 0,C 180,E1 -22250.653,E2 -22250.653} C_VEL
LIN {X 0,Y 287.497,Z 470.628,A -85,B 0,C 180,E1 -22252.661,E2 -22252.661} C_VEL
LIN {X 0,Y 274.979,Z 460.853,A -85,B 0,C 180,E1 -22254.865,E2 -22254.865} C_VEL
LIN {X 0,Y 265.113,Z 452.35,A -85,B 0,C 180,E1 -22256.658,E2 -22256.658} C_VEL
LIN {X 0,Y 255.71,Z 443.207,A -85,B 0,C 180,E1 -22258.42,E2 -22258.42} C_VEL
LIN {X 0,Y 246.423,Z 433.163,A -85,B 0,C 180,E1 -22260.175,E2 -22260.175} C_VEL
LIN {X 0,Y 235.546,Z 420.272,A -85,B 0,C 180,E1 -22262.225,E2 -22262.225} C_VEL
LIN {X 0,Y 225.326,Z 405.329,A -85,B 0,C 180,E1 -22264.456,E2 -22264.456} C_VEL
LIN {X 0,Y 217.744,Z 391.516,A -85,B 0,C 180,E1 -22266.4,E2 -22266.4} C_VEL
LIN {X 0,Y 210.045,Z 375.267,A -85,B 0,C 180,E1 -22268.671,E2 -22268.671} C_VEL
LIN {X 0,Y 203.125,Z 362.313,A -85,B 0,C 180,E1 -22270.855,E2 -22270.855} C_VEL
LIN {X 0,Y 196.139,Z 351.191,A -85,B 0,C 180,E1 -22273.203,E2 -22273.203} C_VEL
LIN {X 0,Y 190.901,Z 343.547,A -85,B 0,C 180,E1 -22275.107,E2 -22275.107} C_VEL
LIN {X 0,Y 188.391,Z 339.72,A -85,B 0,C 180,E1 -22276.091,E2 -22276.091} C_VEL
LIN {X 0,Y 186.402,Z 337.438,A -85,B 0,C 180,E1 -22276.86,E2 -22276.86} C_VEL
LIN {X 0,Y 185.648,Z 335.486,A -85,B 0,C 180,E1 -22277.354,E2 -22277.354} C_VEL
LIN {X 0,Y 185.529,Z 334.907,A -85,B 0,C 180,E1 -22277.931,E2 -22277.931} C_VEL
LIN {X 0,Y 185.555,Z 334.868,A -85,B 0,C 180,E1 -22282.7,E2 -22282.7} C_VEL
LIN {X 0,Y 185.536,Z 334.867,A -85,B 0,C 180,E1 -22287.975,E2 -22287.975} C_VEL
LIN {X 0,Y 185.576,Z 334.846,A -85,B 0,C 180,E1 -22290.577,E2 -22290.577} C_VEL
LIN {X 0,Y 185.582,Z 334.857,A -85,B 0,C 180,E1 -22295.383,E2 -22295.383} C_VEL
LIN {X 0,Y 185.602,Z 334.822,A -85,B 0,C 180,E1 -22300.076,E2 -22300.076} C_VEL
LIN {X 0,Y 185.69,Z 334.853,A -85,B 0,C 180,E1 -22304.638,E2 -22304.638} C_VEL
LIN {X 0,Y 185.884,Z 334.779,A -85,B 0,C 180,E1 -22309.419,E2 -22309.419} C_VEL
LIN {X 0,Y 185.943,Z 334.813,A -85,B 0,C 180,E1 -22313.49,E2 -22313.49} C_VEL
LIN {X 0,Y 186.201,Z 334.748,A -85,B 0,C 180,E1 -22317.838,E2 -22317.838} C_VEL
LIN {X 0,Y 186.4,Z 334.712,A -85,B 0,C 180,E1 -22320.001,E2 -22320.001} C_VEL
LIN {X 0,Y 185.916,Z 334.826,A -85,B 0,C 180,E1 -22324.337,E2 -22324.337} C_VEL
LIN {X 0,Y 185.979,Z 334.767,A -85,B 0,C 180,E1 -22328.695,E2 -22328.695} C_VEL
LIN {X 0,Y 185.725,Z 334.84,A -85,B 0,C 180,E1 -22333.124,E2 -22333.124} C_VEL
LIN {X 0,Y 185.686,Z 334.809,A -85,B 0,C 180,E1 -22337.627,E2 -22337.627} C_VEL
LIN {X 0,Y 185.576,Z 334.864,A -85,B 0,C 180,E1 -22342.255,E2 -22342.255} C_VEL
LIN {X 0,Y 185.556,Z 334.831,A -85,B 0,C 180,E1 -22347.034,E2 -22347.034} C_VEL
LIN {X 0,Y 185.576,Z 334.855,A -85,B 0,C 180,E1 -22349.495,E2 -22349.495} C_VEL
LIN {X 0,Y 185.497,Z 334.849,A -85,B 0,C 180,E1 -22354.634,E2 -22354.634} C_VEL
LIN {X 0,Y 185.475,Z 334.862,A -85,B 0,C 180,E1 -22359.398,E2 -22359.398} C_VEL
LIN {X 0,Y 185.507,Z 335.219,A -85,B 0,C 180,E1 -22360.531,E2 -22360.531} C_VEL
LIN {X 0,Y 186.247,Z 337.867,A -85,B 0,C 180,E1 -22362.629,E2 -22362.629} C_VEL
LIN {X 0,Y 188.85,Z 342.343,A -85,B 0,C 180,E1 -22363.812,E2 -22363.812} C_VEL
LIN {X 0,Y 190.782,Z 345.651,A -85,B 0,C 180,E1 -22364.582,E2 -22364.582} C_VEL
LIN {X 0,Y 195.47,Z 353.722,A -85,B 0,C 180,E1 -22366.353,E2 -22366.353} C_VEL
LIN {X 0,Y 201.447,Z 364.973,A -85,B 0,C 180,E1 -22368.468,E2 -22368.468} C_VEL
LIN {X 0,Y 207.638,Z 378.753,A -85,B 0,C 180,E1 -22370.56,E2 -22370.56} C_VEL
LIN {X 0,Y 210.615,Z 386.589,A -85,B 0,C 180,E1 -22371.552,E2 -22371.552} C_VEL
LIN {X 0,Y 212.68,Z 400.794,A -85,B 0,C 180,E1 -22372.582,E2 -22372.582} C_VEL
LIN {X 0,Y 210.462,Z 444.967,A -85,B 0,C 180,E1 -22374.042,E2 -22374.042} C_VEL
LIN {X 0,Y 209.252,Z 456.153,A -85,B 0,C 180,E1 -22374.633,E2 -22374.633} C_VEL
LIN {X 0,Y 207.143,Z 469.362,A -85,B 0,C 180,E1 -22375.664,E2 -22375.664} C_VEL
LIN {X 0,Y 204.622,Z 480.905,A -85,B 0,C 180,E1 -22376.959,E2 -22376.959} C_VEL
LIN {X 0,Y 202.346,Z 490.178,A -85,B 0,C 180,E1 -22378.31,E2 -22378.31} C_VEL
LIN {X 0,Y 199.751,Z 499.117,A -85,B 0,C 180,E1 -22379.91,E2 -22379.91} C_VEL
LIN {X 0,Y 197.028,Z 507.642,A -85,B 0,C 180,E1 -22381.796,E2 -22381.796} C_VEL
LIN {X 0,Y 194.551,Z 514.857,A -85,B 0,C 180,E1 -22383.736,E2 -22383.736} C_VEL
LIN {X 0,Y 192.357,Z 521.058,A -85,B 0,C 180,E1 -22385.731,E2 -22385.731} C_VEL
LIN {X 0,Y 190.067,Z 527.598,A -85,B 0,C 180,E1 -22388.299,E2 -22388.299} C_VEL
LIN {X 0,Y 188.346,Z 532.099,A -85,B 0,C 180,E1 -22390.378,E2 -22390.378} C_VEL
LIN {X 0,Y 186.192,Z 537.589,A -85,B 0,C 180,E1 -22393.555,E2 -22393.555} C_VEL
LIN {X 0,Y 184.71,Z 541.918,A -85,B 0,C 180,E1 -22396.804,E2 -22396.804} C_VEL
LIN {X 0,Y 184.046,Z 544.076,A -85,B 0,C 180,E1 -22398.787,E2 -22398.787} C_VEL
LIN {X 0,Y 182.964,Z 545.726,A -85,B 0,C 180,E1 -22400.526,E2 -22400.526} C_VEL
LIN {X 0,Y 179.68,Z 547.67,A -85,B 0,C 180,E1 -22403.419,E2 -22403.419} C_VEL
LIN {X 0,Y 177.107,Z 548.581,A -85,B 0,C 180,E1 -22405.834,E2 -22405.834} C_VEL
LIN {X 0,Y 176.045,Z 548.957,A -85,B 0,C 180,E1 -22407.734,E2 -22407.734} C_VEL
LIN {X 0,Y 175.968,Z 548.996,A -85,B 0,C 180,E1 -22408.381,E2 -22408.381} C_VEL
LIN {X 0,Y 176.058,Z 549.108,A -85,B 0,C 180,E1 -22410,E2 -22410} C_VEL
LIN {X 0,Y 175.951,Z 548.756,A -85,B 0,C 180,E1 -22413.037,E2 -22413.037} C_VEL
LIN {X 0,Y 176.118,Z 547.291,A -85,B 0,C 180,E1 -22416.876,E2 -22416.876} C_VEL
LIN {X 0,Y 176.46,Z 545.898,A -85,B 0,C 180,E1 -22419.167,E2 -22419.167} C_VEL
LIN {X 0,Y 177.35,Z 542.942,A -85,B 0,C 180,E1 -22422.589,E2 -22422.589} C_VEL
LIN {X 0,Y 178.713,Z 538.948,A -85,B 0,C 180,E1 -22425.978,E2 -22425.978} C_VEL
LIN {X 0,Y 180.849,Z 533.82,A -85,B 0,C 180,E1 -22429.288,E2 -22429.288} C_VEL
LIN {X 0,Y 182.994,Z 528.559,A -85,B 0,C 180,E1 -22431.99,E2 -22431.99} C_VEL
LIN {X 0,Y 184.991,Z 523.293,A -85,B 0,C 180,E1 -22434.244,E2 -22434.244} C_VEL
LIN {X 0,Y 187.574,Z 516.289,A -85,B 0,C 180,E1 -22436.718,E2 -22436.718} C_VEL
LIN {X 0,Y 190.102,Z 509.365,A -85,B 0,C 180,E1 -22438.724,E2 -22438.724} C_VEL
LIN {X 0,Y 192.888,Z 501.191,A -85,B 0,C 180,E1 -22440.67,E2 -22440.67} C_VEL
LIN {X 0,Y 195.53,Z 492.685,A -85,B 0,C 180,E1 -22442.32,E2 -22442.32} C_VEL
LIN {X 0,Y 197.932,Z 483.975,A -85,B 0,C 180,E1 -22443.696,E2 -22443.696} C_VEL
LIN {X 0,Y 200.17,Z 474.219,A -85,B 0,C 180,E1 -22444.94,E2 -22444.94} C_VEL
LIN {X 0,Y 201.974,Z 465.432,A -85,B 0,C 180,E1 -22445.803,E2 -22445.803} C_VEL
LIN {X 0,Y 203.636,Z 455.065,A -85,B 0,C 180,E1 -22446.575,E2 -22446.575} C_VEL
LIN {X 0,Y 204.707,Z 445.077,A -85,B 0,C 180,E1 -22447.115,E2 -22447.115} C_VEL
LIN {X 0,Y 206.486,Z 413.494,A -85,B 0,C 180,E1 -22448.184,E2 -22448.184} C_VEL
LIN {X 0,Y 206.934,Z 400.867,A -85,B 0,C 180,E1 -22448.633,E2 -22448.633} C_VEL
LIN {X 0,Y 204.946,Z 388.216,A -85,B 0,C 180,E1 -22449.636,E2 -22449.636} C_VEL
LIN {X 0,Y 199.525,Z 375.02,A -85,B 0,C 180,E1 -22451.546,E2 -22451.546} C_VEL
LIN {X 0,Y 194.005,Z 363.479,A -85,B 0,C 180,E1 -22453.57,E2 -22453.57} C_VEL
LIN {X 0,Y 187.372,Z 351.506,A -85,B 0,C 180,E1 -22456.161,E2 -22456.161} C_VEL
LIN {X 0,Y 184.756,Z 347.122,A -85,B 0,C 180,E1 -22457.251,E2 -22457.251} C_VEL
LIN {X 0,Y 181.662,Z 342.165,A -85,B 0,C 180,E1 -22458.599,E2 -22458.599} C_VEL
LIN {X 0,Y 179.203,Z 338.297,A -85,B 0,C 180,E1 -22459.767,E2 -22459.767} C_VEL
LIN {X 0,Y 178.701,Z 337.084,A -85,B 0,C 180,E1 -22460.275,E2 -22460.275} C_VEL
LIN {X 0,Y 178.405,Z 335.8,A -85,B 0,C 180,E1 -22461.55,E2 -22461.55} C_VEL
LIN {X 0,Y 178.484,Z 335.721,A -85,B 0,C 180,E1 -22466.545,E2 -22466.545} C_VEL
LIN {X 0,Y 178.521,Z 335.742,A -85,B 0,C 180,E1 -22470.006,E2 -22470.006} C_VEL
LIN {X 0,Y 178.518,Z 335.716,A -85,B 0,C 180,E1 -22474.884,E2 -22474.884} C_VEL
LIN {X 0,Y 178.619,Z 335.687,A -85,B 0,C 180,E1 -22480.785,E2 -22480.785} C_VEL
LIN {X 0,Y 178.653,Z 335.727,A -85,B 0,C 180,E1 -22486.346,E2 -22486.346} C_VEL
LIN {X 0,Y 178.908,Z 335.645,A -85,B 0,C 180,E1 -22490.958,E2 -22490.958} C_VEL
LIN {X 0,Y 178.864,Z 335.706,A -85,B 0,C 180,E1 -22495.492,E2 -22495.492} C_VEL
LIN {X 0,Y 179.363,Z 335.587,A -85,B 0,C 180,E1 -22499.999,E2 -22499.999} C_VEL
LIN {X 0,Y 178.862,Z 335.702,A -85,B 0,C 180,E1 -22504.506,E2 -22504.506} C_VEL
LIN {X 0,Y 178.907,Z 335.649,A -85,B 0,C 180,E1 -22509.039,E2 -22509.039} C_VEL
LIN {X 0,Y 178.652,Z 335.723,A -85,B 0,C 180,E1 -22513.651,E2 -22513.651} C_VEL
LIN {X 0,Y 178.618,Z 335.689,A -85,B 0,C 180,E1 -22519.215,E2 -22519.215} C_VEL
LIN {X 0,Y 178.52,Z 335.726,A -85,B 0,C 180,E1 -22525.116,E2 -22525.116} C_VEL
LIN {X 0,Y 178.493,Z 335.751,A -85,B 0,C 180,E1 -22530.786,E2 -22530.786} C_VEL
LIN {X 0,Y 178.479,Z 335.723,A -85,B 0,C 180,E1 -22534.218,E2 -22534.218} C_VEL
LIN {X 0,Y 178.506,Z 335.887,A -85,B 0,C 180,E1 -22539.774,E2 -22539.774} C_VEL
LIN {X 0,Y 178.741,Z 336.876,A -85,B 0,C 180,E1 -22540.355,E2 -22540.355} C_VEL
LIN {X 0,Y 180.365,Z 339.708,A -85,B 0,C 180,E1 -22541.173,E2 -22541.173} C_VEL
LIN {X 0,Y 182.003,Z 341.337,A -85,B 0,C 180,E1 -22541.858,E2 -22541.858} C_VEL
LIN {X 0,Y 184.202,Z 344.715,A -85,B 0,C 180,E1 -22542.812,E2 -22542.812} C_VEL
LIN {X 0,Y 185.446,Z 346.299,A -85,B 0,C 180,E1 -22543.316,E2 -22543.316} C_VEL
LIN {X 0,Y 193.1,Z 357.672,A -85,B 0,C 180,E1 -22546.267,E2 -22546.267} C_VEL
LIN {X 0,Y 200.721,Z 370.476,A -85,B 0,C 180,E1 -22548.927,E2 -22548.927} C_VEL
LIN {X 0,Y 207.942,Z 384.833,A -85,B 0,C 180,E1 -22551.277,E2 -22551.277} C_VEL
LIN {X 0,Y 216.258,Z 402.365,A -85,B 0,C 180,E1 -22553.747,E2 -22553.747} C_VEL
LIN {X 0,Y 224.517,Z 416.048,A -85,B 0,C 180,E1 -22555.809,E2 -22555.809} C_VEL
LIN {X 0,Y 232.961,Z 427.74,A -85,B 0,C 180,E1 -22557.639,E2 -22557.639} C_VEL
LIN {X 0,Y 243.473,Z 440.261,A -85,B 0,C 180,E1 -22559.785,E2 -22559.785} C_VEL
LIN {X 0,Y 254.504,Z 452.074,A -85,B 0,C 180,E1 -22562.085,E2 -22562.085} C_VEL
LIN {X 0,Y 266.631,Z 463.211,A -85,B 0,C 180,E1 -22564.523,E2 -22564.523} C_VEL
LIN {X 0,Y 280.012,Z 473.817,A -85,B 0,C 180,E1 -22567.068,E2 -22567.068} C_VEL
LIN {X 0,Y 292.747,Z 483.178,A -85,B 0,C 180,E1 -22569.432,E2 -22569.432} C_VEL
LIN {X 0,Y 300.156,Z 488.679,A -85,B 0,C 180,E1 -22570.865,E2 -22570.865} C_VEL
LIN {X 0,Y 307.418,Z 493.76,A -85,B 0,C 180,E1 -22572.42,E2 -22572.42} C_VEL
LIN {X 0,Y 314.193,Z 498.653,A -85,B 0,C 180,E1 -22574.118,E2 -22574.118} C_VEL
LIN {X 0,Y 321.081,Z 503.236,A -85,B 0,C 180,E1 -22576.068,E2 -22576.068} C_VEL
LIN {X 0,Y 325.839,Z 506.069,A -85,B 0,C 180,E1 -22577.544,E2 -22577.544} C_VEL
LIN {X 0,Y 331.132,Z 509.839,A -85,B 0,C 180,E1 -22579.668,E2 -22579.668} C_VEL
LIN {X 0,Y 335.089,Z 512.4,A -85,B 0,C 180,E1 -22581.558,E2 -22581.558} C_VEL
LIN {X 0,Y 337.434,Z 513.686,A -85,B 0,C 180,E1 -22582.821,E2 -22582.821} C_VEL
LIN {X 0,Y 339.447,Z 514.662,A -85,B 0,C 180,E1 -22584.058,E2 -22584.058} C_VEL
LIN {X 0,Y 341.108,Z 515.401,A -85,B 0,C 180,E1 -22585.273,E2 -22585.273} C_VEL
LIN {X 0,Y 342.473,Z 515.87,A -85,B 0,C 180,E1 -22586.47,E2 -22586.47} C_VEL
LIN {X 0,Y 343.327,Z 516.25,A -85,B 0,C 180,E1 -22587.654,E2 -22587.654} C_VEL
LIN {X 0,Y 343.816,Z 516.483,A -85,B 0,C 180,E1 -22588.829,E2 -22588.829} C_VEL
LIN {X 0,Y 344.062,Z 516.487,A -85,B 0,C 180,E1 -22590,E2 -22590} C_VEL
LIN {X 0,Y 343.845,Z 516.446,A -85,B 0,C 180,E1 -22591.171,E2 -22591.171} C_VEL
LIN {X 0,Y 343.352,Z 516.206,A -85,B 0,C 180,E1 -22592.346,E2 -22592.346} C_VEL
LIN {X 0,Y 342.459,Z 515.849,A -85,B 0,C 180,E1 -22593.53,E2 -22593.53} C_VEL
LIN {X 0,Y 341.113,Z 515.36,A -85,B 0,C 180,E1 -22594.727,E2 -22594.727} C_VEL
LIN {X 0,Y 339.232,Z 514.574,A -85,B 0,C 180,E1 -22596.056,E2 -22596.056} C_VEL
LIN {X 0,Y 337.42,Z 513.67,A -85,B 0,C 180,E1 -22597.179,E2 -22597.179} C_VEL
LIN {X 0,Y 334.292,Z 511.912,A -85,B 0,C 180,E1 -22598.851,E2 -22598.851} C_VEL
LIN {X 0,Y 331.127,Z 509.857,A -85,B 0,C 180,E1 -22600.326,E2 -22600.326} C_VEL
LIN {X 0,Y 325.811,Z 506.074,A -85,B 0,C 180,E1 -22602.457,E2 -22602.457} C_VEL
LIN {X 0,Y 319.338,Z 502.068,A -85,B 0,C 180,E1 -22604.457,E2 -22604.457} C_VEL
LIN {X 0,Y 314.207,Z 498.596,A -85,B 0,C 180,E1 -22605.891,E2 -22605.891} C_VEL
LIN {X 0,Y 307.451,Z 493.819,A -85,B 0,C 180,E1 -22607.57,E2 -22607.57} C_VEL
LIN {X 0,Y 300.194,Z 488.705,A -85,B 0,C 180,E1 -22609.132,E2 -22609.132} C_VEL
LIN {X 0,Y 292.752,Z 483.158,A -85,B 0,C 180,E1 -22610.57,E2 -22610.57} C_VEL
LIN {X 0,Y 280.02,Z 473.787,A -85,B 0,C 180,E1 -22612.935,E2 -22612.935} C_VEL
LIN {X 0,Y 268.002,Z 464.277,A -85,B 0,C 180,E1 -22615.217,E2 -22615.217} C_VEL
LIN {X 0,Y 255.838,Z 453.414,A -85,B 0,C 180,E1 -22617.637,E2 -22617.637} C_VEL
LIN {X 0,Y 244.635,Z 441.578,A -85,B 0,C 180,E1 -22619.965,E2 -22619.965} C_VEL
LIN {X 0,Y 235.685,Z 431.099,A -85,B 0,C 180,E1 -22621.806,E2 -22621.806} C_VEL
LIN {X 0,Y 226.934,Z 419.617,A -85,B 0,C 180,E1 -22623.641,E2 -22623.641} C_VEL
LIN {X 0,Y 218.108,Z 405.686,A -85,B 0,C 180,E1 -22625.763,E2 -22625.763} C_VEL
LIN {X 0,Y 210.916,Z 391.436,A -85,B 0,C 180,E1 -22627.793,E2 -22627.793} C_VEL
LIN {X 0,Y 204.596,Z 378.021,A -85,B 0,C 180,E1 -22629.788,E2 -22629.788} C_VEL
LIN {X 0,Y 198.475,Z 366.516,A -85,B 0,C 180,E1 -22631.833,E2 -22631.833} C_VEL
LIN {X 0,Y 190.565,Z 353.72,A -85,B 0,C 180,E1 -22634.677,E2 -22634.677} C_VEL
LIN {X 0,Y 184.474,Z 344.996,A -85,B 0,C 180,E1 -22637.081,E2 -22637.081} C_VEL
LIN {X 0,Y 182.126,Z 341.596,A -85,B 0,C 180,E1 -22638.084,E2 -22638.084} C_VEL
LIN {X 0,Y 181.343,Z 340.593,A -85,B 0,C 180,E1 -22638.42,E2 -22638.42} C_VEL
LIN {X 0,Y 179.425,Z 338.372,A -85,B 0,C 180,E1 -22639.254,E2 -22639.254} C_VEL
LIN {X 0,Y 178.584,Z 336.286,A -85,B 0,C 180,E1 -22639.879,E2 -22639.879} C_VEL
LIN {X 0,Y 178.474,Z 335.78,A -85,B 0,C 180,E1 -22640.584,E2 -22640.584} C_VEL
LIN {X 0,Y 178.479,Z 335.723,A -85,B 0,C 180,E1 -22645.782,E2 -22645.782} C_VEL
LIN {X 0,Y 178.517,Z 335.733,A -85,B 0,C 180,E1 -22650.008,E2 -22650.008} C_VEL
LIN {X 0,Y 178.52,Z 335.726,A -85,B 0,C 180,E1 -22654.884,E2 -22654.884} C_VEL
LIN {X 0,Y 178.618,Z 335.689,A -85,B 0,C 180,E1 -22660.785,E2 -22660.785} C_VEL
LIN {X 0,Y 178.652,Z 335.723,A -85,B 0,C 180,E1 -22666.349,E2 -22666.349} C_VEL
LIN {X 0,Y 178.907,Z 335.649,A -85,B 0,C 180,E1 -22670.961,E2 -22670.961} C_VEL
LIN {X 0,Y 178.862,Z 335.702,A -85,B 0,C 180,E1 -22675.494,E2 -22675.494} C_VEL
LIN {X 0,Y 179.363,Z 335.587,A -85,B 0,C 180,E1 -22680.001,E2 -22680.001} C_VEL
LIN {X 0,Y 178.864,Z 335.706,A -85,B 0,C 180,E1 -22684.508,E2 -22684.508} C_VEL
LIN {X 0,Y 178.908,Z 335.645,A -85,B 0,C 180,E1 -22689.042,E2 -22689.042} C_VEL
LIN {X 0,Y 178.653,Z 335.727,A -85,B 0,C 180,E1 -22693.654,E2 -22693.654} C_VEL
LIN {X 0,Y 178.619,Z 335.687,A -85,B 0,C 180,E1 -22699.215,E2 -22699.215} C_VEL
LIN {X 0,Y 178.518,Z 335.716,A -85,B 0,C 180,E1 -22705.116,E2 -22705.116} C_VEL
LIN {X 0,Y 178.498,Z 335.751,A -85,B 0,C 180,E1 -22710.788,E2 -22710.788} C_VEL
LIN {X 0,Y 178.483,Z 335.721,A -85,B 0,C 180,E1 -22714.22,E2 -22714.22} C_VEL
LIN {X 0,Y 178.512,Z 335.945,A -85,B 0,C 180,E1 -22718.739,E2 -22718.739} C_VEL
LIN {X 0,Y 178.932,Z 337.639,A -85,B 0,C 180,E1 -22720.03,E2 -22720.03} C_VEL
LIN {X 0,Y 181.269,Z 341.693,A -85,B 0,C 180,E1 -22721.233,E2 -22721.233} C_VEL
LIN {X 0,Y 182.946,Z 344.155,A -85,B 0,C 180,E1 -22721.966,E2 -22721.966} C_VEL
LIN {X 0,Y 186.343,Z 349.745,A -85,B 0,C 180,E1 -22723.414,E2 -22723.414} C_VEL
LIN {X 0,Y 191.751,Z 359.372,A -85,B 0,C 180,E1 -22725.58,E2 -22725.58} C_VEL
LIN {X 0,Y 197.052,Z 369.618,A -85,B 0,C 180,E1 -22727.558,E2 -22727.558} C_VEL
LIN {X 0,Y 202.75,Z 382.599,A -85,B 0,C 180,E1 -22729.597,E2 -22729.597} C_VEL
LIN {X 0,Y 205.273,Z 389.492,A -85,B 0,C 180,E1 -22730.496,E2 -22730.496} C_VEL
LIN {X 0,Y 207.033,Z 402.254,A -85,B 0,C 180,E1 -22731.449,E2 -22731.449} C_VEL
LIN {X 0,Y 204.774,Z 444.228,A -85,B 0,C 180,E1 -22732.844,E2 -22732.844} C_VEL
LIN {X 0,Y 203.636,Z 455.063,A -85,B 0,C 180,E1 -22733.425,E2 -22733.425} C_VEL
LIN {X 0,Y 202.029,Z 465.434,A -85,B 0,C 180,E1 -22734.208,E2 -22734.208} C_VEL
LIN {X 0,Y 199.82,Z 476.235,A -85,B 0,C 180,E1 -22735.297,E2 -22735.297} C_VEL
LIN {X 0,Y 196.716,Z 488.633,A -85,B 0,C 180,E1 -22736.988,E2 -22736.988} C_VEL
LIN {X 0,Y 193.618,Z 498.922,A -85,B 0,C 180,E1 -22738.853,E2 -22738.853} C_VEL
LIN {X 0,Y 190.798,Z 507.448,A -85,B 0,C 180,E1 -22740.788,E2 -22740.788} C_VEL
LIN {X 0,Y 188.176,Z 514.662,A -85,B 0,C 180,E1 -22742.774,E2 -22742.774} C_VEL
LIN {X 0,Y 185.886,Z 520.863,A -85,B 0,C 180,E1 -22744.828,E2 -22744.828} C_VEL
LIN {X 0,Y 183.466,Z 527.403,A -85,B 0,C 180,E1 -22747.477,E2 -22747.477} C_VEL
LIN {X 0,Y 181.621,Z 531.903,A -85,B 0,C 180,E1 -22749.619,E2 -22749.619} C_VEL
LIN {X 0,Y 179.372,Z 537.395,A -85,B 0,C 180,E1 -22752.911,E2 -22752.911} C_VEL
LIN {X 0,Y 177.768,Z 541.724,A -85,B 0,C 180,E1 -22756.279,E2 -22756.279} C_VEL
LIN {X 0,Y 176.989,Z 544.115,A -85,B 0,C 180,E1 -22758.575,E2 -22758.575} C_VEL
LIN {X 0,Y 176.465,Z 545.898,A -85,B 0,C 180,E1 -22760.834,E2 -22760.834} C_VEL
LIN {X 0,Y 176.01,Z 548.356,A -85,B 0,C 180,E1 -22765.42,E2 -22765.42} C_VEL
LIN {X 0,Y 175.968,Z 548.996,A -85,B 0,C 180,E1 -22768.381,E2 -22768.381} C_VEL
LIN {X 0,Y 175.296,Z 549.105,A -85,B 0,C 180,E1 -22770.29,E2 -22770.29} C_VEL
LIN {X 0,Y 173.69,Z 548.925,A -85,B 0,C 180,E1 -22772.169,E2 -22772.169} C_VEL
LIN {X 0,Y 170.053,Z 547.704,A -85,B 0,C 180,E1 -22775.967,E2 -22775.967} C_VEL
LIN {X 0,Y 169.201,Z 546.543,A -85,B 0,C 180,E1 -22778.273,E2 -22778.273} C_VEL
LIN {X 0,Y 169.234,Z 546.256,A -85,B 0,C 180,E1 -22778.605,E2 -22778.605} C_VEL
LIN {X 0,Y 170.023,Z 543.9,A -85,B 0,C 180,E1 -22781.927,E2 -22781.927} C_VEL
LIN {X 0,Y 171.3,Z 540.285,A -85,B 0,C 180,E1 -22785.466,E2 -22785.466} C_VEL
LIN {X 0,Y 173.323,Z 535.54,A -85,B 0,C 180,E1 -22788.928,E2 -22788.928} C_VEL
LIN {X 0,Y 175.899,Z 529.519,A -85,B 0,C 180,E1 -22792.306,E2 -22792.306} C_VEL
LIN {X 0,Y 178.234,Z 523.786,A -85,B 0,C 180,E1 -22794.914,E2 -22794.914} C_VEL
LIN {X 0,Y 180.621,Z 517.721,A -85,B 0,C 180,E1 -22797.206,E2 -22797.206} C_VEL
LIN {X 0,Y 183.9,Z 509.171,A -85,B 0,C 180,E1 -22799.789,E2 -22799.789} C_VEL
LIN {X 0,Y 186.816,Z 500.997,A -85,B 0,C 180,E1 -22801.781,E2 -22801.781} C_VEL
LIN {X 0,Y 189.565,Z 492.491,A -85,B 0,C 180,E1 -22803.468,E2 -22803.468} C_VEL
LIN {X 0,Y 192.06,Z 483.781,A -85,B 0,C 180,E1 -22804.872,E2 -22804.872} C_VEL
LIN {X 0,Y 194.401,Z 474.026,A -85,B 0,C 180,E1 -22806.137,E2 -22806.137} C_VEL
LIN {X 0,Y 196.271,Z 465.239,A -85,B 0,C 180,E1 -22807.013,E2 -22807.013} C_VEL
LIN {X 0,Y 197.988,Z 454.691,A -85,B 0,C 180,E1 -22807.814,E2 -22807.814} C_VEL
LIN {X 0,Y 199.141,Z 444.439,A -85,B 0,C 180,E1 -22808.363,E2 -22808.363} C_VEL
LIN {X 0,Y 201.451,Z 402.583,A -85,B 0,C 180,E1 -22809.804,E2 -22809.804} C_VEL
LIN {X 0,Y 199.715,Z 391.13,A -85,B 0,C 180,E1 -22810.747,E2 -22810.747} C_VEL
LIN {X 0,Y 194.662,Z 378.662,A -85,B 0,C 180,E1 -22812.639,E2 -22812.639} C_VEL
LIN {X 0,Y 189.673,Z 367.977,A -85,B 0,C 180,E1 -22814.586,E2 -22814.586} C_VEL
LIN {X 0,Y 183.334,Z 356.26,A -85,B 0,C 180,E1 -22817.214,E2 -22817.214} C_VEL
LIN {X 0,Y 180.634,Z 351.757,A -85,B 0,C 180,E1 -22818.404,E2 -22818.404} C_VEL
LIN {X 0,Y 177.857,Z 347.187,A -85,B 0,C 180,E1 -22819.692,E2 -22819.692} C_VEL
LIN {X 0,Y 174.68,Z 342.291,A -85,B 0,C 180,E1 -22821.241,E2 -22821.241} C_VEL
LIN {X 0,Y 172.04,Z 338.854,A -85,B 0,C 180,E1 -22822.578,E2 -22822.578} C_VEL
LIN {X 0,Y 171.451,Z 337.203,A -85,B 0,C 180,E1 -22823.164,E2 -22823.164} C_VEL
LIN {X 0,Y 171.4,Z 336.679,A -85,B 0,C 180,E1 -22823.882,E2 -22823.882} C_VEL
LIN {X 0,Y 171.455,Z 336.629,A -85,B 0,C 180,E1 -22829.404,E2 -22829.404} C_VEL
LIN {X 0,Y 171.457,Z 336.59,A -85,B 0,C 180,E1 -22834.39,E2 -22834.39} C_VEL
LIN {X 0,Y 171.575,Z 336.563,A -85,B 0,C 180,E1 -22840.87,E2 -22840.87} C_VEL
LIN {X 0,Y 171.572,Z 336.611,A -85,B 0,C 180,E1 -22845.771,E2 -22845.771} C_VEL
LIN {X 0,Y 171.845,Z 336.523,A -85,B 0,C 180,E1 -22850.583,E2 -22850.583} C_VEL
LIN {X 0,Y 171.812,Z 336.584,A -85,B 0,C 180,E1 -22855.306,E2 -22855.306} C_VEL
LIN {X 0,Y 172.326,Z 336.463,A -85,B 0,C 180,E1 -22859.999,E2 -22859.999} C_VEL
LIN {X 0,Y 171.811,Z 336.582,A -85,B 0,C 180,E1 -22864.691,E2 -22864.691} C_VEL
LIN {X 0,Y 171.843,Z 336.526,A -85,B 0,C 180,E1 -22869.414,E2 -22869.414} C_VEL
LIN {X 0,Y 171.571,Z 336.612,A -85,B 0,C 180,E1 -22874.226,E2 -22874.226} C_VEL
LIN {X 0,Y 171.539,Z 336.57,A -85,B 0,C 180,E1 -22879.56,E2 -22879.56} C_VEL
LIN {X 0,Y 171.457,Z 336.598,A -85,B 0,C 180,E1 -22885.61,E2 -22885.61} C_VEL
LIN {X 0,Y 171.451,Z 336.623,A -85,B 0,C 180,E1 -22890.594,E2 -22890.594} C_VEL
LIN {X 0,Y 171.436,Z 336.681,A -85,B 0,C 180,E1 -22896.744,E2 -22896.744} C_VEL
LIN {X 0,Y 171.586,Z 337.511,A -85,B 0,C 180,E1 -22897.442,E2 -22897.442} C_VEL
